RoboDK station: Example-03.d-Polishing Canadian Canoe - KUKA.rdk

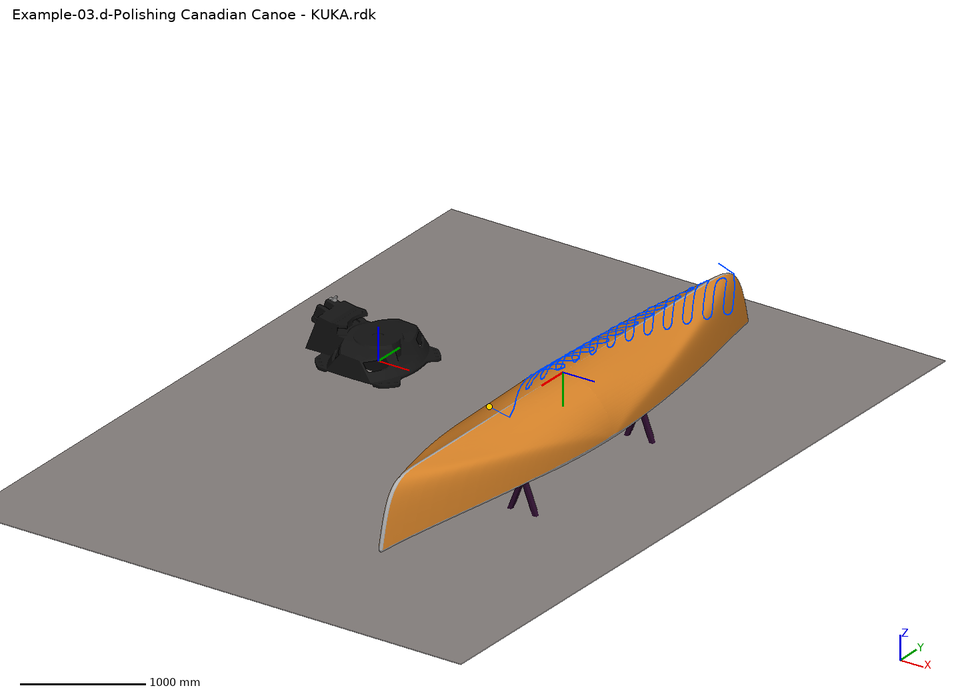
[picture v0: the station drawn from its stored meshes, robots at their saved joint values, targets as dots, program paths as lines]
Station Canoe Record Station final. Poses are relative to the parent item; angles as X-Y-Z fixed-axis rotations.
  - frame World at (0, 0, 0) mm
    - object Floor at (1290, -760, -10) mm, rotated rx 0 ry 0 rz 90 deg, size 6720 x 4800 x 9.6 mm, geometry from Floor.step
    - object Canoe Holder at (2372.71, -1561.9, -4.29) mm, rotated rx -180 ry 0 rz 0 deg, size 378 x 1657.8 x 756 mm, geometry from Canoe Holder.step
  - frame KUKA KR 100 R3500 press Base at (0, 0, 0) mm
    - robot KUKA KR 100 R3500 press: 6 axes, payload 100 kg, reach 3501 mm, repeatability 0.06 mm, weight 1240 kg
        joint limits [-185, -120, -120, -350, -122.5, -350] to [185, 70, 155, 350, 122.5, 350]; home [0, -90, 90, 0, 0, 0]; saved at [6.556, -77.694, 99.787, -0.648, 50.095, 7.142]
      - tool Sanding Tool, TCP at (0, 0, 140.65) mm, size 253.6 x 268.9 x 140.8 mm, geometry from Sanding Tool.step
  - frame Part at (2500, -1000, 1000) mm, rotated rx -90 ry 0 rz -90 deg
    - object Canadian Canoe at (0, 0, 0) mm, size 5096.7 x 583.7 x 963.7 mm, geometry from Canadian Canoe.step
    - object Polish Path 1 at (0, 0, 0) mm
  - machining project Polish Path 1 Settings: rotZ(0) | rotX(0)*rotY(0) | rotz(0) | ChangeTool(toolid) | onPathStart | PolishOn | onPoint | PolishOff | onFinish | SetRPM(%1) | SetTool(%1) | Extruder(%1) | default | default | OutOnMov(%1) | OutOffMov(%1) | onPathFinish | M_RunCode(%1)
  - program Polish (1259 instructions, listed below)
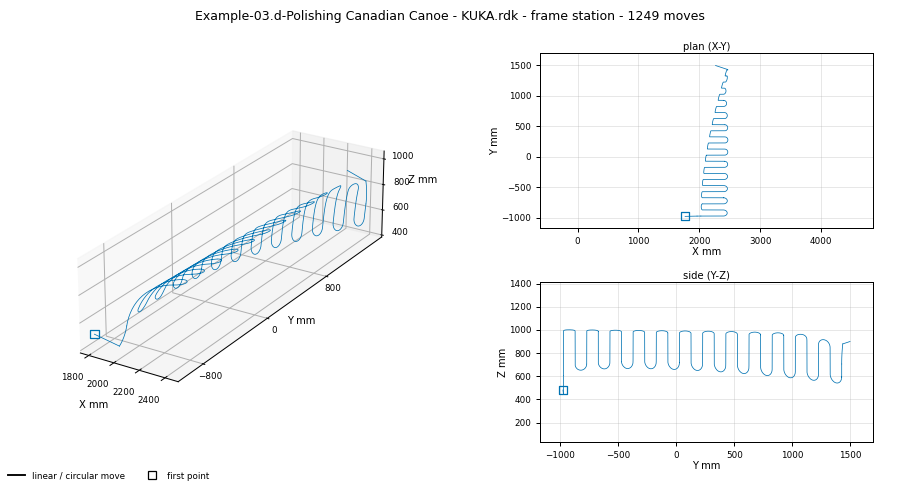
[picture p0: tool path of Example-03.d-Polishing Canadian Canoe - KUKA.rdk in frame station, 1249 of 1249 moves have a stored position in this frame; points joined in program order, loops and branches not executed]

--- program Polish (robot KUKA KR 100 R3500 press) ---
  Call ChangeTool(toolid)
  Smooth(1)
  Set Ref.: Part
  Set Tool: Sanding Tool
  Show Sanding Tool
  Set speed (200.0 mm/s)
  MoveJ 1 to (-21.87, 518.76, -734.4) mm, rotated rx 0 ry 10.84 rz 96.44 deg; joints [35.321, -70.266, 137.679, -138.31, 61.6, 158.371]
  MoveL 2 to (-21.87, 518.76, -734.4) mm, rotated rx 0 ry 10.84 rz 96.44 deg; joints [35.321, -70.266, 137.679, -138.31, 61.6, 158.371]
  Call PolishOn
  MoveL 3 to (-26.09, 556.13, -537.97) mm, rotated rx 0 ry 10.84 rz 96.44 deg; joints [31.728, -64.525, 130.322, -141.639, 59.446, 158.433]
  MoveC 4 to (-26.54, 477.64, -500.08) mm, rotated rx 0 ry 10.84 rz 96.44 deg; joints [31.115, -67.789, 128.968, -140.477, 55.681, 155.246] to (-26.66, 393.76, -476.39) mm, rotated rx 0 ry 10.84 rz 96.44 deg; joints [30.747, -71.291, 127.887, -138.729, 52.066, 151.749]
  MoveL 5 to (-26.66, 393.76, -476.39) mm, rotated rx 0 ry 10.84 rz 96.44 deg; joints [30.747, -71.291, 127.887, -138.729, 52.066, 151.749]
  MoveL 6 to (-26.66, 393.76, -476.39) mm, rotated rx 0 ry 10.84 rz 96.44 deg; joints [30.747, -71.291, 127.887, -138.729, 52.066, 151.749]
  Set speed (50.0 mm/s)
  MoveL 7 to (-26.66, 376.38, -472.76) mm, rotated rx 0 ry 12.85 rz 94.05 deg; joints [30.597, -72.582, 127.559, -137.347, 48.797, 152.34]
  MoveL 8 to (-26.66, 359.15, -468.51) mm, rotated rx 0 ry 14.9 rz 92.45 deg; joints [30.438, -73.793, 127.144, -135.658, 45.564, 151.886]
  MoveL 9 to (-26.66, 342.08, -463.65) mm, rotated rx 0 ry 16.96 rz 91.33 deg; joints [30.267, -74.917, 126.648, -133.634, 42.392, 150.663]
  MoveL 10 to (-26.66, 325.2, -458.16) mm, rotated rx 0 ry 19.04 rz 90.51 deg; joints [30.085, -75.951, 126.072, -131.226, 39.302, 148.785]
  MoveL 11 to (-26.66, 308.53, -452.07) mm, rotated rx 0 ry 21.12 rz 89.91 deg; joints [29.892, -76.889, 125.421, -128.37, 36.321, 146.284]
  MoveL 12 to (-26.66, 292.1, -445.38) mm, rotated rx 0 ry 23.2 rz 89.45 deg; joints [29.688, -77.729, 124.697, -124.985, 33.477, 143.138]
  MoveL 13 to (-26.66, 275.92, -438.09) mm, rotated rx 0 ry 25.28 rz 89.1 deg; joints [29.473, -78.472, 123.903, -120.973, 30.8, 139.286]
  MoveL 14 to (-26.66, 260.02, -430.23) mm, rotated rx 0 ry 27.37 rz 88.83 deg; joints [29.249, -79.115, 123.044, -116.23, 28.333, 134.648]
  MoveL 15 to (-26.66, 244.43, -421.8) mm, rotated rx 0 ry 29.45 rz 88.63 deg; joints [29.016, -79.659, 122.123, -110.659, 26.129, 129.146]
  MoveL 16 to (-26.66, 229.18, -412.82) mm, rotated rx 0 ry 31.53 rz 88.47 deg; joints [28.774, -80.105, 121.144, -104.187, 24.244, 122.718]
  MoveL 17 to (-26.66, 214.28, -403.3) mm, rotated rx 0 ry 33.61 rz 88.36 deg; joints [28.526, -80.455, 120.109, -96.804, 22.741, 115.363]
  MoveL 18 to (-26.66, 199.73, -393.26) mm, rotated rx 0 ry 35.69 rz 88.29 deg; joints [28.27, -80.711, 119.022, -88.615, 21.681, 107.193]
  MoveL 19 to (-26.66, 185.57, -382.7) mm, rotated rx 0 ry 37.76 rz 88.24 deg; joints [28.009, -80.875, 117.885, -79.876, 21.113, 98.467]
  MoveL 20 to (-26.66, 171.8, -371.63) mm, rotated rx 0 ry 39.84 rz 88.21 deg; joints [27.742, -80.951, 116.702, -70.965, 21.059, 89.568]
  MoveL 21 to (-26.66, 158.43, -360.06) mm, rotated rx 0 ry 41.92 rz 88.2 deg; joints [27.471, -80.94, 115.473, -62.307, 21.506, 80.922]
  MoveL 22 to (-26.66, 145.48, -348.01) mm, rotated rx 0 ry 44 rz 88.21 deg; joints [27.195, -80.847, 114.201, -54.254, 22.41, 72.884]
  MoveL 23 to (-26.66, 132.96, -335.48) mm, rotated rx 0 ry 46.08 rz 88.23 deg; joints [26.916, -80.673, 112.889, -47.021, 23.705, 65.671]
  MoveL 24 to (-26.66, 120.89, -322.49) mm, rotated rx 0 ry 48.17 rz 88.26 deg; joints [26.634, -80.422, 111.538, -40.68, 25.319, 59.356]
  MoveL 25 to (-26.66, 109.3, -309.06) mm, rotated rx 0 ry 50.26 rz 88.31 deg; joints [26.35, -80.098, 110.152, -35.208, 27.184, 53.915]
  MoveL 26 to (-26.66, 98.22, -295.23) mm, rotated rx 0 ry 52.34 rz 88.36 deg; joints [26.065, -79.703, 108.734, -30.523, 29.238, 49.268]
  MoveL 27 to (-26.66, 87.66, -281.03) mm, rotated rx 0 ry 54.43 rz 88.42 deg; joints [25.78, -79.242, 107.288, -26.513, 31.434, 45.305]
  MoveL 28 to (-26.66, 77.63, -266.46) mm, rotated rx 0 ry 56.51 rz 88.49 deg; joints [25.495, -78.717, 105.814, -23.071, 33.738, 41.916]
  MoveL 29 to (-26.66, 68.14, -251.54) mm, rotated rx 0 ry 58.59 rz 88.56 deg; joints [25.211, -78.131, 104.313, -20.1, 36.12, 39.008]
  MoveL 30 to (-26.66, 59.2, -236.29) mm, rotated rx 0 ry 60.67 rz 88.64 deg; joints [24.928, -77.488, 102.788, -17.519, 38.562, 36.499]
  MoveL 31 to (-26.66, 50.82, -220.71) mm, rotated rx 0 ry 62.76 rz 88.72 deg; joints [24.646, -76.789, 101.238, -15.262, 41.049, 34.323]
  MoveL 32 to (-26.66, 43.01, -204.84) mm, rotated rx 0 ry 64.84 rz 88.81 deg; joints [24.365, -76.038, 99.664, -13.273, 43.568, 32.426]
  MoveL 33 to (-26.66, 35.77, -188.67) mm, rotated rx 0 ry 66.93 rz 88.9 deg; joints [24.087, -75.236, 98.069, -11.508, 46.112, 30.763]
  MoveL 34 to (-26.66, 29.12, -172.23) mm, rotated rx 0 ry 69.03 rz 88.99 deg; joints [23.811, -74.386, 96.451, -9.931, 48.674, 29.299]
  MoveL 35 to (-26.66, 23.07, -155.55) mm, rotated rx 0 ry 71.12 rz 89.09 deg; joints [23.539, -73.49, 94.814, -8.515, 51.247, 28.008]
  MoveL 36 to (-26.66, 17.65, -138.69) mm, rotated rx 0 ry 73.21 rz 89.19 deg; joints [23.27, -72.554, 93.162, -7.236, 53.821, 26.866]
  MoveL 37 to (-26.66, 12.84, -121.65) mm, rotated rx 0 ry 75.3 rz 89.29 deg; joints [23.005, -71.578, 91.496, -6.073, 56.395, 25.853]
  MoveL 38 to (-26.66, 8.67, -104.47) mm, rotated rx 0 ry 77.39 rz 89.39 deg; joints [22.744, -70.564, 89.814, -5.01, 58.966, 24.952]
  MoveL 39 to (-26.66, 8.67, -104.47) mm, rotated rx 0 ry 77.39 rz 89.39 deg; joints [22.744, -70.564, 89.814, -5.01, 58.966, 24.952]
  MoveL 40 to (-27.51, 6.41, -93.75) mm, rotated rx 0 ry 78.68 rz 89.45 deg; joints [22.566, -69.932, 88.785, -4.39, 60.546, 24.425]
  MoveL 41 to (-30.02, 4.45, -83.22) mm, rotated rx 0 ry 79.94 rz 89.51 deg; joints [22.359, -69.329, 87.813, -3.806, 62.065, 23.908]
  MoveL 42 to (-34.12, 2.8, -73.18) mm, rotated rx 0 ry 81.12 rz 89.56 deg; joints [22.129, -68.772, 86.925, -3.274, 63.484, 23.411]
  MoveL 43 to (-39.8, 1.48, -63.88) mm, rotated rx 0 ry 82.19 rz 89.6 deg; joints [21.88, -68.28, 86.145, -2.802, 64.765, 22.939]
  MoveL 44 to (-43.22, 0.94, -59.64) mm, rotated rx 0 ry 82.68 rz 89.62 deg; joints [21.751, -68.066, 85.808, -2.593, 65.337, 22.715]
  MoveL 45 to (-47.01, 0.48, -55.73) mm, rotated rx 0 ry 83.12 rz 89.64 deg; joints [21.618, -67.878, 85.512, -2.405, 65.854, 22.499]
  MoveL 46 to (-51.17, 0.09, -52.22) mm, rotated rx 0 ry 83.51 rz 89.65 deg; joints [21.485, -67.72, 85.263, -2.24, 66.307, 22.295]
  MoveL 47 to (-55.67, -0.22, -49.18) mm, rotated rx 0 ry 83.85 rz 89.67 deg; joints [21.351, -67.597, 85.069, -2.099, 66.686, 22.102]
  MoveL 48 to (-60.51, -0.46, -46.68) mm, rotated rx 0 ry 84.11 rz 89.67 deg; joints [21.219, -67.513, 84.934, -1.984, 66.981, 21.922]
  MoveL 49 to (-65.61, -0.62, -44.79) mm, rotated rx 0 ry 84.3 rz 89.68 deg; joints [21.089, -67.474, 84.867, -1.899, 67.181, 21.759]
  MoveL 50 to (-70.92, -0.71, -43.6) mm, rotated rx 0 ry 84.4 rz 89.68 deg; joints [20.965, -67.482, 84.872, -1.845, 67.278, 21.614]
  MoveL 51 to (-76.36, -0.72, -43.15) mm, rotated rx 0 ry 84.42 rz 89.67 deg; joints [20.847, -67.54, 84.952, -1.823, 67.264, 21.49]
  MoveL 52 to (-81.8, -0.66, -43.46) mm, rotated rx 0 ry 84.34 rz 89.66 deg; joints [20.74, -67.648, 85.106, -1.833, 67.137, 21.389]
  MoveL 53 to (-87.14, -0.52, -44.52) mm, rotated rx 0 ry 84.17 rz 89.65 deg; joints [20.643, -67.803, 85.332, -1.873, 66.903, 21.312]
  MoveL 54 to (-92.3, -0.3, -46.28) mm, rotated rx 0 ry 83.92 rz 89.62 deg; joints [20.56, -68, 85.622, -1.941, 66.568, 21.261]
  MoveL 55 to (-97.19, -0.01, -48.67) mm, rotated rx 0 ry 83.6 rz 89.6 deg; joints [20.49, -68.234, 85.967, -2.035, 66.143, 21.236]
  MoveL 56 to (-101.76, 0.37, -51.62) mm, rotated rx 0 ry 83.21 rz 89.57 deg; joints [20.432, -68.498, 86.359, -2.151, 65.641, 21.234]
  MoveL 57 to (-105.99, 0.82, -55.04) mm, rotated rx 0 ry 82.77 rz 89.53 deg; joints [20.388, -68.786, 86.79, -2.287, 65.073, 21.257]
  MoveL 58 to (-109.84, 1.36, -58.88) mm, rotated rx 0 ry 82.29 rz 89.49 deg; joints [20.357, -69.093, 87.252, -2.441, 64.45, 21.302]
  MoveL 59 to (-113.32, 1.98, -63.07) mm, rotated rx 0 ry 81.76 rz 89.45 deg; joints [20.338, -69.415, 87.739, -2.611, 63.78, 21.37]
  MoveL 60 to (-119.09, 3.46, -72.25) mm, rotated rx 0 ry 80.62 rz 89.36 deg; joints [20.334, -70.086, 88.764, -2.994, 62.336, 21.568]
  MoveL 61 to (-123.26, 5.27, -82.23) mm, rotated rx 0 ry 79.41 rz 89.27 deg; joints [20.374, -70.773, 89.829, -3.428, 60.794, 21.85]
  MoveL 62 to (-125.8, 7.38, -92.7) mm, rotated rx 0 ry 78.14 rz 89.17 deg; joints [20.457, -71.455, 90.903, -3.911, 59.199, 22.212]
  MoveL 63 to (-126.66, 9.76, -103.38) mm, rotated rx 0 ry 76.86 rz 89.08 deg; joints [20.58, -72.113, 91.96, -4.437, 57.594, 22.653]
  MoveL 64 to (-126.66, 9.76, -103.38) mm, rotated rx 0 ry 76.86 rz 89.08 deg; joints [20.58, -72.113, 91.96, -4.437, 57.594, 22.653]
  MoveL 65 to (-126.66, 17.22, -131.53) mm, rotated rx 0 ry 73.48 rz 88.86 deg; joints [20.967, -73.761, 94.694, -6.011, 53.356, 24.056]
  MoveL 66 to (-126.66, 26.34, -159.24) mm, rotated rx 0 ry 70.1 rz 88.67 deg; joints [21.365, -75.303, 97.386, -7.878, 49.121, 25.774]
  MoveL 67 to (-126.66, 37.07, -186.38) mm, rotated rx 0 ry 66.74 rz 88.5 deg; joints [21.775, -76.728, 100.027, -10.127, 44.908, 27.89]
  MoveL 68 to (-126.66, 49.36, -212.8) mm, rotated rx 0 ry 63.4 rz 88.36 deg; joints [22.195, -78.024, 102.61, -12.882, 40.74, 30.524]
  MoveL 69 to (-126.66, 63.15, -238.44) mm, rotated rx 0 ry 60.06 rz 88.26 deg; joints [22.623, -79.183, 105.132, -16.314, 36.644, 33.846]
  MoveL 70 to (-126.66, 78.41, -263.23) mm, rotated rx 0 ry 56.73 rz 88.19 deg; joints [23.059, -80.193, 107.588, -20.673, 32.668, 38.1]
  MoveL 71 to (-126.66, 95.1, -287.12) mm, rotated rx 0 ry 53.42 rz 88.17 deg; joints [23.501, -81.043, 109.974, -26.314, 28.89, 43.635]
  MoveL 72 to (-126.66, 113.18, -310.05) mm, rotated rx 0 ry 50.1 rz 88.21 deg; joints [23.948, -81.719, 112.284, -33.726, 25.435, 50.931]
  MoveL 73 to (-126.66, 132.55, -331.89) mm, rotated rx 0 ry 46.8 rz 88.32 deg; joints [24.398, -82.205, 114.505, -43.444, 22.513, 60.518]
  MoveL 74 to (-126.66, 153.11, -352.55) mm, rotated rx 0 ry 43.5 rz 88.51 deg; joints [24.847, -82.489, 116.626, -55.814, 20.415, 72.728]
  MoveL 75 to (-126.66, 174.81, -371.99) mm, rotated rx 0 ry 40.22 rz 88.81 deg; joints [25.293, -82.556, 118.64, -70.412, 19.477, 87.12]
  MoveL 76 to (-126.66, 197.6, -390.16) mm, rotated rx 0 ry 36.95 rz 89.25 deg; joints [25.735, -82.393, 120.536, -85.632, 19.933, 102.065]
  MoveL 77 to (-126.66, 221.41, -407.03) mm, rotated rx 0 ry 33.68 rz 89.87 deg; joints [26.17, -81.987, 122.306, -99.424, 21.768, 115.479]
  MoveL 78 to (-126.66, 246.16, -422.53) mm, rotated rx 0 ry 30.43 rz 90.72 deg; joints [26.595, -81.327, 123.935, -110.611, 24.74, 126.138]
  MoveL 79 to (-126.66, 271.73, -436.59) mm, rotated rx 0 ry 27.19 rz 91.88 deg; joints [27.005, -80.405, 125.409, -119.146, 28.539, 133.925]
  MoveL 80 to (-126.66, 298.05, -449.17) mm, rotated rx 0 ry 23.97 rz 93.45 deg; joints [27.397, -79.22, 126.718, -125.536, 32.912, 139.252]
  MoveL 81 to (-126.66, 298.05, -449.17) mm, rotated rx 0 ry 23.97 rz 93.45 deg; joints [27.397, -79.22, 126.718, -125.536, 32.912, 139.252]
  MoveL 82 to (-127.57, 307.4, -453.24) mm, rotated rx 0 ry 22.87 rz 94.13 deg; joints [27.505, -78.761, 127.15, -127.373, 34.523, 140.591]
  MoveL 83 to (-130.27, 316.51, -457.06) mm, rotated rx 0 ry 21.82 rz 94.91 deg; joints [27.562, -78.32, 127.583, -129.005, 36.088, 141.626]
  MoveL 84 to (-134.68, 325.06, -460.55) mm, rotated rx 0 ry 20.87 rz 95.71 deg; joints [27.561, -77.916, 128.01, -130.458, 37.553, 142.427]
  MoveL 85 to (-140.71, 332.73, -463.63) mm, rotated rx 0 ry 19.99 rz 96.43 deg; joints [27.5, -77.568, 128.431, -131.809, 38.881, 143.152]
  MoveL 86 to (-144.29, 336.12, -464.99) mm, rotated rx 0 ry 19.57 rz 96.71 deg; joints [27.445, -77.419, 128.64, -132.482, 39.488, 143.56]
  MoveL 87 to (-148.2, 339.15, -466.21) mm, rotated rx 0 ry 19.15 rz 96.9 deg; joints [27.372, -77.288, 128.85, -133.177, 40.06, 144.046]
  MoveL 88 to (-152.44, 341.79, -467.28) mm, rotated rx 0 ry 18.73 rz 96.99 deg; joints [27.282, -77.177, 129.06, -133.911, 40.6, 144.643]
  MoveL 89 to (-156.95, 344, -468.2) mm, rotated rx 0 ry 18.31 rz 96.96 deg; joints [27.174, -77.084, 129.272, -134.688, 41.108, 145.369]
  MoveL 90 to (-161.69, 345.73, -468.95) mm, rotated rx 0 ry 17.88 rz 96.8 deg; joints [27.051, -77.014, 129.481, -135.496, 41.579, 146.218]
  MoveL 91 to (-166.61, 346.96, -469.52) mm, rotated rx 0 ry 17.46 rz 96.53 deg; joints [26.913, -76.969, 129.683, -136.309, 42, 147.154]
  MoveL 92 to (-171.65, 347.66, -469.91) mm, rotated rx 0 ry 17.09 rz 96.18 deg; joints [26.765, -76.954, 129.872, -137.083, 42.346, 148.113]
  MoveL 93 to (-176.74, 347.81, -470.12) mm, rotated rx 0 ry 16.8 rz 95.79 deg; joints [26.61, -76.976, 130.039, -137.76, 42.582, 149.006]
  MoveL 94 to (-181.84, 347.4, -470.15) mm, rotated rx 0 ry 16.61 rz 95.41 deg; joints [26.452, -77.042, 130.179, -138.295, 42.677, 149.752]
  MoveL 95 to (-186.86, 346.44, -470) mm, rotated rx 0 ry 16.56 rz 95.08 deg; joints [26.294, -77.157, 130.285, -138.647, 42.603, 150.279]
  MoveL 96 to (-191.75, 344.95, -469.68) mm, rotated rx 0 ry 16.67 rz 94.83 deg; joints [26.14, -77.321, 130.355, -138.794, 42.346, 150.54]
  MoveL 97 to (-196.44, 342.96, -469.2) mm, rotated rx 0 ry 16.92 rz 94.67 deg; joints [25.992, -77.532, 130.385, -138.725, 41.904, 150.518]
  MoveL 98 to (-200.89, 340.51, -468.56) mm, rotated rx 0 ry 17.33 rz 94.6 deg; joints [25.851, -77.786, 130.377, -138.441, 41.29, 150.216]
  MoveL 99 to (-205.06, 337.66, -467.76) mm, rotated rx 0 ry 17.86 rz 94.6 deg; joints [25.717, -78.075, 130.33, -137.951, 40.524, 149.658]
  MoveL 100 to (-212.46, 330.89, -465.7) mm, rotated rx 0 ry 19.23 rz 94.73 deg; joints [25.472, -78.721, 130.131, -136.411, 38.646, 147.908]
  MoveL 101 to (-218.45, 323.03, -463.03) mm, rotated rx 0 ry 20.86 rz 94.87 deg; joints [25.253, -79.402, 129.811, -134.269, 36.508, 145.573]
  MoveL 102 to (-222.9, 314.4, -459.75) mm, rotated rx 0 ry 22.54 rz 94.9 deg; joints [25.059, -80.059, 129.399, -131.722, 34.323, 142.947]
  MoveL 103 to (-225.67, 305.32, -455.94) mm, rotated rx 0 ry 24.16 rz 94.76 deg; joints [24.891, -80.653, 128.925, -128.966, 32.247, 140.254]
  MoveL 104 to (-226.66, 296.05, -451.69) mm, rotated rx 0 ry 25.64 rz 94.48 deg; joints [24.753, -81.164, 128.41, -126.131, 30.355, 137.613]
  MoveL 105 to (-226.66, 296.05, -451.69) mm, rotated rx 0 ry 25.64 rz 94.48 deg; joints [24.753, -81.164, 128.41, -126.131, 30.355, 137.613]
  MoveL 106 to (-226.66, 270.18, -438.28) mm, rotated rx 0 ry 29.16 rz 93.21 deg; joints [24.38, -82.288, 126.92, -117.969, 25.867, 130.316]
  MoveL 107 to (-226.66, 245.16, -423.4) mm, rotated rx 0 ry 32.32 rz 91.9 deg; joints [23.966, -83.105, 125.374, -108.343, 22.255, 121.554]
  MoveL 108 to (-226.66, 221.07, -407.26) mm, rotated rx 0 ry 35.36 rz 90.79 deg; joints [23.538, -83.661, 123.728, -96.225, 19.574, 110.144]
  MoveL 109 to (-226.66, 197.82, -389.81) mm, rotated rx 0 ry 38.4 rz 89.91 deg; joints [23.104, -83.977, 121.962, -81.528, 18.063, 96]
  MoveL 110 to (-226.66, 175.5, -371.14) mm, rotated rx 0 ry 41.45 rz 89.24 deg; joints [22.669, -84.067, 120.08, -65.719, 17.94, 80.615]
  MoveL 111 to (-226.66, 154.2, -351.29) mm, rotated rx 0 ry 44.51 rz 88.74 deg; joints [22.236, -83.94, 118.092, -51.11, 19.167, 66.33]
  MoveL 112 to (-226.66, 134.01, -330.36) mm, rotated rx 0 ry 47.59 rz 88.38 deg; joints [21.807, -83.612, 116.007, -39.179, 21.459, 54.645]
  MoveL 113 to (-226.66, 114.99, -308.38) mm, rotated rx 0 ry 50.69 rz 88.14 deg; joints [21.385, -83.094, 113.834, -30.079, 24.47, 45.735]
  MoveL 114 to (-226.66, 97.2, -285.42) mm, rotated rx 0 ry 53.8 rz 88 deg; joints [20.97, -82.4, 111.579, -23.269, 27.933, 39.072]
  MoveL 115 to (-226.66, 80.67, -261.51) mm, rotated rx 0 ry 56.93 rz 87.94 deg; joints [20.565, -81.541, 109.247, -18.143, 31.677, 34.061]
  MoveL 116 to (-226.66, 65.47, -236.71) mm, rotated rx 0 ry 60.09 rz 87.96 deg; joints [20.168, -80.528, 106.841, -14.214, 35.601, 30.228]
  MoveL 117 to (-226.66, 51.64, -211.07) mm, rotated rx 0 ry 63.27 rz 88.03 deg; joints [19.782, -79.372, 104.366, -11.151, 39.636, 27.249]
  MoveL 118 to (-226.66, 39.23, -184.63) mm, rotated rx 0 ry 66.48 rz 88.16 deg; joints [19.406, -78.081, 101.827, -8.724, 43.736, 24.898]
  MoveL 119 to (-226.66, 28.33, -157.54) mm, rotated rx 0 ry 69.69 rz 88.34 deg; joints [19.044, -76.67, 99.236, -6.78, 47.865, 23.026]
  MoveL 120 to (-226.66, 18.99, -129.94) mm, rotated rx 0 ry 72.93 rz 88.56 deg; joints [18.696, -75.147, 96.597, -5.195, 52.015, 21.515]
  MoveL 121 to (-226.66, 11.24, -101.9) mm, rotated rx 0 ry 76.19 rz 88.82 deg; joints [18.36, -73.52, 93.91, -3.883, 56.181, 20.285]
  MoveL 122 to (-226.66, 11.24, -101.9) mm, rotated rx 0 ry 76.19 rz 88.82 deg; joints [18.36, -73.52, 93.91, -3.883, 56.181, 20.285]
  MoveL 123 to (-227.52, 8.78, -91.34) mm, rotated rx 0 ry 77.4 rz 88.93 deg; joints [18.22, -72.9, 92.915, -3.447, 57.721, 19.867]
  MoveL 124 to (-230.03, 6.62, -80.99) mm, rotated rx 0 ry 78.57 rz 89.03 deg; joints [18.048, -72.307, 91.971, -3.043, 59.197, 19.449]
  MoveL 125 to (-234.15, 4.79, -71.12) mm, rotated rx 0 ry 79.66 rz 89.13 deg; joints [17.849, -71.758, 91.106, -2.682, 60.569, 19.04]
  MoveL 126 to (-239.84, 3.29, -62.01) mm, rotated rx 0 ry 80.65 rz 89.22 deg; joints [17.628, -71.271, 90.345, -2.369, 61.796, 18.645]
  MoveL 127 to (-243.26, 2.67, -57.85) mm, rotated rx 0 ry 81.09 rz 89.26 deg; joints [17.511, -71.059, 90.014, -2.234, 62.338, 18.455]
  MoveL 128 to (-247.05, 2.13, -54.03) mm, rotated rx 0 ry 81.48 rz 89.3 deg; joints [17.39, -70.872, 89.724, -2.113, 62.823, 18.27]
  MoveL 129 to (-251.2, 1.68, -50.61) mm, rotated rx 0 ry 81.82 rz 89.34 deg; joints [17.266, -70.715, 89.479, -2.009, 63.243, 18.092]
  MoveL 130 to (-255.68, 1.31, -47.64) mm, rotated rx 0 ry 82.11 rz 89.37 deg; joints [17.139, -70.591, 89.285, -1.923, 63.589, 17.922]
  MoveL 131 to (-260.49, 1.03, -45.2) mm, rotated rx 0 ry 82.33 rz 89.39 deg; joints [17.012, -70.504, 89.148, -1.854, 63.852, 17.761]
  MoveL 132 to (-265.54, 0.83, -43.36) mm, rotated rx 0 ry 82.47 rz 89.41 deg; joints [16.886, -70.46, 89.074, -1.804, 64.022, 17.61]
  MoveL 133 to (-270.8, 0.73, -42.18) mm, rotated rx 0 ry 82.54 rz 89.42 deg; joints [16.762, -70.46, 89.067, -1.773, 64.092, 17.472]
  MoveL 134 to (-276.18, 0.72, -41.71) mm, rotated rx 0 ry 82.53 rz 89.42 deg; joints [16.642, -70.507, 89.131, -1.761, 64.058, 17.349]
  MoveL 135 to (-281.57, 0.81, -41.96) mm, rotated rx 0 ry 82.43 rz 89.41 deg; joints [16.528, -70.601, 89.264, -1.768, 63.918, 17.242]
  MoveL 136 to (-286.88, 1, -42.92) mm, rotated rx 0 ry 82.25 rz 89.39 deg; joints [16.423, -70.739, 89.464, -1.792, 63.677, 17.153]
  MoveL 137 to (-291.99, 1.28, -44.55) mm, rotated rx 0 ry 82 rz 89.36 deg; joints [16.328, -70.916, 89.724, -1.833, 63.343, 17.083]
  MoveL 138 to (-296.87, 1.66, -46.8) mm, rotated rx 0 ry 81.68 rz 89.33 deg; joints [16.244, -71.128, 90.036, -1.887, 62.927, 17.032]
  MoveL 139 to (-301.46, 2.13, -49.6) mm, rotated rx 0 ry 81.31 rz 89.28 deg; joints [16.17, -71.37, 90.396, -1.954, 62.436, 17]
  MoveL 140 to (-305.71, 2.7, -52.88) mm, rotated rx 0 ry 80.88 rz 89.23 deg; joints [16.108, -71.637, 90.794, -2.033, 61.884, 16.986]
  MoveL 141 to (-309.61, 3.36, -56.58) mm, rotated rx 0 ry 80.42 rz 89.18 deg; joints [16.057, -71.922, 91.223, -2.122, 61.28, 16.992]
  MoveL 142 to (-313.12, 4.12, -60.63) mm, rotated rx 0 ry 79.92 rz 89.12 deg; joints [16.017, -72.223, 91.677, -2.22, 60.634, 17.015]
  MoveL 143 to (-318.97, 5.89, -69.57) mm, rotated rx 0 ry 78.86 rz 89 deg; joints [15.97, -72.854, 92.64, -2.443, 59.244, 17.116]
  MoveL 144 to (-323.21, 7.99, -79.34) mm, rotated rx 0 ry 77.72 rz 88.86 deg; joints [15.966, -73.504, 93.645, -2.702, 57.769, 17.287]
  MoveL 145 to (-325.79, 10.39, -89.6) mm, rotated rx 0 ry 76.56 rz 88.73 deg; joints [16.005, -74.152, 94.663, -2.995, 56.253, 17.529]
  MoveL 146 to (-326.66, 13.03, -100.1) mm, rotated rx 0 ry 75.39 rz 88.61 deg; joints [16.087, -74.781, 95.668, -3.324, 54.732, 17.842]
  MoveL 147 to (-326.66, 13.03, -100.1) mm, rotated rx 0 ry 75.39 rz 88.61 deg; joints [16.087, -74.781, 95.668, -3.324, 54.732, 17.842]
  MoveL 148 to (-326.66, 21.62, -129.56) mm, rotated rx 0 ry 72.14 rz 88.3 deg; joints [16.384, -76.457, 98.434, -4.419, 50.483, 18.938]
  MoveL 149 to (-326.66, 31.86, -158.52) mm, rotated rx 0 ry 68.93 rz 88.05 deg; joints [16.696, -78.02, 101.142, -5.79, 46.265, 20.303]
  MoveL 150 to (-326.66, 43.68, -186.84) mm, rotated rx 0 ry 65.77 rz 87.87 deg; joints [17.024, -79.46, 103.785, -7.521, 42.095, 22.014]
  MoveL 151 to (-326.66, 57.07, -214.48) mm, rotated rx 0 ry 62.61 rz 87.76 deg; joints [17.37, -80.777, 106.377, -9.76, 37.937, 24.211]
  MoveL 152 to (-326.66, 71.99, -241.41) mm, rotated rx 0 ry 59.46 rz 87.73 deg; joints [17.731, -81.959, 108.912, -12.681, 33.824, 27.066]
  MoveL 153 to (-326.66, 88.43, -267.6) mm, rotated rx 0 ry 56.34 rz 87.78 deg; joints [18.11, -82.994, 111.386, -16.559, 29.804, 30.844]
  MoveL 154 to (-326.66, 106.3, -292.91) mm, rotated rx 0 ry 53.25 rz 87.94 deg; joints [18.503, -83.867, 113.783, -21.795, 25.967, 35.936]
  MoveL 155 to (-326.66, 125.5, -317.22) mm, rotated rx 0 ry 50.19 rz 88.22 deg; joints [18.91, -84.564, 116.098, -28.995, 22.426, 42.935]
  MoveL 156 to (-326.66, 145.96, -340.48) mm, rotated rx 0 ry 47.16 rz 88.64 deg; joints [19.33, -85.073, 118.326, -38.968, 19.38, 52.635]
  MoveL 157 to (-326.66, 167.61, -362.62) mm, rotated rx 0 ry 44.14 rz 89.22 deg; joints [19.761, -85.38, 120.461, -52.426, 17.151, 65.732]
  MoveL 158 to (-326.66, 190.17, -383.4) mm, rotated rx 0 ry 41.15 rz 89.97 deg; joints [20.197, -85.471, 122.48, -68.918, 16.152, 81.766]
  MoveL 159 to (-326.66, 201.28, -392.87) mm, rotated rx 0 ry 39.72 rz 90.38 deg; joints [20.406, -85.435, 123.41, -77.359, 16.195, 89.951]
  MoveL 160 to (-326.66, 212.12, -401.66) mm, rotated rx 0 ry 38.32 rz 90.81 deg; joints [20.605, -85.35, 124.282, -85.411, 16.568, 97.738]
  MoveL 161 to (-326.66, 222.63, -409.76) mm, rotated rx 0 ry 36.96 rz 91.23 deg; joints [20.794, -85.221, 125.101, -92.845, 17.223, 104.906]
  MoveL 162 to (-326.66, 232.74, -417.18) mm, rotated rx 0 ry 35.62 rz 91.63 deg; joints [20.97, -85.053, 125.869, -99.575, 18.105, 111.38]
  MoveL 163 to (-326.66, 242.39, -423.92) mm, rotated rx 0 ry 34.28 rz 91.99 deg; joints [21.131, -84.849, 126.591, -105.63, 19.166, 117.202]
  MoveL 164 to (-326.66, 251.51, -429.98) mm, rotated rx 0 ry 32.92 rz 92.29 deg; joints [21.274, -84.614, 127.272, -111.099, 20.372, 122.48]
  MoveL 165 to (-326.66, 260.05, -435.37) mm, rotated rx 0 ry 31.53 rz 92.48 deg; joints [21.4, -84.35, 127.917, -116.095, 21.703, 127.341]
  MoveL 166 to (-326.66, 268.03, -440.12) mm, rotated rx 0 ry 30.09 rz 92.56 deg; joints [21.506, -84.056, 128.534, -120.728, 23.159, 131.917]
  MoveL 167 to (-326.66, 275.46, -444.29) mm, rotated rx 0 ry 28.57 rz 92.5 deg; joints [21.592, -83.733, 129.125, -125.047, 24.738, 136.271]
  MoveL 168 to (-326.66, 282.36, -447.93) mm, rotated rx 0 ry 26.99 rz 92.29 deg; joints [21.66, -83.377, 129.693, -129.092, 26.453, 140.459]
  MoveL 169 to (-326.66, 282.36, -447.93) mm, rotated rx 0 ry 26.99 rz 92.29 deg; joints [21.66, -83.377, 129.693, -129.092, 26.453, 140.459]
  MoveL 170 to (-326.94, 287.31, -450.39) mm, rotated rx 0 ry 25.72 rz 92 deg; joints [21.69, -83.085, 130.119, -132.038, 27.859, 143.599]
  MoveL 171 to (-327.75, 292.26, -452.71) mm, rotated rx 0 ry 24.31 rz 91.56 deg; joints [21.696, -82.758, 130.567, -135.044, 29.444, 146.906]
  MoveL 172 to (-329.09, 297.17, -454.86) mm, rotated rx 0 ry 22.79 rz 90.94 deg; joints [21.675, -82.391, 131.03, -138.048, 31.215, 150.347]
  MoveL 173 to (-330.91, 301.99, -456.81) mm, rotated rx 0 ry 21.17 rz 90.13 deg; joints [21.629, -81.985, 131.495, -140.95, 33.145, 153.847]
  MoveL 174 to (-333.19, 306.67, -458.54) mm, rotated rx 0 ry 19.51 rz 89.1 deg; joints [21.559, -81.545, 131.948, -143.66, 35.189, 157.333]
  MoveL 175 to (-335.89, 311.18, -460.04) mm, rotated rx 0 ry 17.87 rz 87.87 deg; joints [21.468, -81.081, 132.376, -146.107, 37.277, 160.742]
  MoveL 176 to (-339.01, 315.49, -461.32) mm, rotated rx 0 ry 16.31 rz 86.47 deg; joints [21.36, -80.611, 132.768, -148.25, 39.327, 164.022]
  MoveL 177 to (-342.49, 319.53, -462.37) mm, rotated rx 0 ry 14.88 rz 84.94 deg; joints [21.237, -80.153, 133.117, -150.077, 41.257, 167.129]
  MoveL 178 to (-346.31, 323.27, -463.21) mm, rotated rx 0 ry 13.41 rz 82.89 deg; joints [21.091, -79.668, 133.453, -151.867, 43.277, 170.673]
  MoveL 179 to (-350.44, 326.66, -463.83) mm, rotated rx 0 ry 12.04 rz 80.41 deg; joints [20.928, -79.194, 133.758, -153.486, 45.22, 174.47]
  MoveL 180 to (-354.87, 329.66, -464.26) mm, rotated rx 0 ry 10.88 rz 77.74 deg; joints [20.757, -78.771, 134.016, -154.834, 46.912, 178.199]
  MoveL 181 to (-359.55, 332.21, -464.52) mm, rotated rx 0 ry 9.96 rz 75.08 deg; joints [20.58, -78.419, 134.232, -155.932, 48.306, 181.702]
  MoveL 182 to (-364.46, 334.24, -464.62) mm, rotated rx 0 ry 9.26 rz 72.59 deg; joints [20.399, -78.147, 134.409, -156.818, 49.395, 184.844]
  MoveL 183 to (-369.53, 335.7, -464.58) mm, rotated rx 0 ry 8.77 rz 70.44 deg; joints [20.217, -77.959, 134.555, -157.528, 50.19, 187.5]
  MoveL 184 to (-374.71, 336.52, -464.42) mm, rotated rx 0 ry 8.45 rz 68.72 deg; joints [20.035, -77.853, 134.673, -158.093, 50.717, 189.594]
  MoveL 185 to (-379.92, 336.69, -464.16) mm, rotated rx 0 ry 8.28 rz 67.52 deg; joints [19.855, -77.827, 134.768, -158.535, 50.994, 191.069]
  MoveL 186 to (-385.04, 336.19, -463.81) mm, rotated rx 0 ry 8.23 rz 66.87 deg; joints [19.681, -77.878, 134.839, -158.866, 51.039, 191.904]
  MoveL 187 to (-389.95, 335.08, -463.38) mm, rotated rx 0 ry 8.3 rz 66.76 deg; joints [19.516, -77.998, 134.887, -159.091, 50.874, 192.117]
  MoveL 188 to (-394.58, 333.42, -462.88) mm, rotated rx 0 ry 8.48 rz 67.13 deg; joints [19.364, -78.18, 134.914, -159.216, 50.515, 191.764]
  MoveL 189 to (-398.93, 331.27, -462.33) mm, rotated rx 0 ry 8.76 rz 67.94 deg; joints [19.222, -78.419, 134.918, -159.242, 49.972, 190.901]
  MoveL 190 to (-406.78, 325.7, -461.04) mm, rotated rx 0 ry 9.65 rz 70.64 deg; joints [18.976, -79.057, 134.856, -158.971, 48.317, 187.834]
  MoveL 191 to (-413.38, 318.81, -459.48) mm, rotated rx 0 ry 11.07 rz 74.34 deg; joints [18.782, -79.891, 134.678, -158.164, 45.857, 183.333]
  MoveL 192 to (-418.72, 310.96, -457.58) mm, rotated rx 0 ry 13.15 rz 78.48 deg; joints [18.642, -80.899, 134.349, -156.611, 42.506, 177.789]
  MoveL 193 to (-422.83, 302.26, -455.17) mm, rotated rx 0 ry 16 rz 82.45 deg; joints [18.55, -82.04, 133.819, -153.972, 38.224, 171.452]
  MoveL 194 to (-425.56, 292.93, -452.13) mm, rotated rx 0 ry 19.24 rz 85.44 deg; joints [18.485, -83.146, 133.108, -150.269, 33.608, 165.089]
  MoveL 195 to (-426.36, 287.77, -450.23) mm, rotated rx 0 ry 20.9 rz 86.51 deg; joints [18.455, -83.66, 132.692, -148.031, 31.313, 161.924]
  MoveL 196 to (-426.66, 282.26, -448.03) mm, rotated rx 0 ry 22.74 rz 87.55 deg; joints [18.437, -84.169, 132.197, -145.135, 28.867, 158.176]
  MoveL 197 to (-426.66, 282.26, -448.03) mm, rotated rx 0 ry 22.74 rz 87.55 deg; joints [18.437, -84.169, 132.197, -145.135, 28.867, 158.176]
  MoveL 198 to (-426.66, 270.66, -442.69) mm, rotated rx 0 ry 26.62 rz 89.24 deg; joints [18.397, -85.071, 131.045, -137.33, 24.077, 149.056]
  MoveL 199 to (-426.66, 267.36, -441) mm, rotated rx 0 ry 27.67 rz 89.6 deg; joints [18.379, -85.282, 130.705, -134.713, 22.867, 146.175]
  MoveL 200 to (-426.66, 263.49, -438.92) mm, rotated rx 0 ry 28.88 rz 89.96 deg; joints [18.354, -85.506, 130.302, -131.423, 21.548, 142.627]
  MoveL 201 to (-426.66, 259.04, -436.39) mm, rotated rx 0 ry 30.19 rz 90.29 deg; joints [18.32, -85.73, 129.84, -127.389, 20.184, 138.36]
  MoveL 202 to (-426.66, 254.01, -433.38) mm, rotated rx 0 ry 31.58 rz 90.58 deg; joints [18.274, -85.946, 129.323, -122.561, 18.841, 133.338]
  MoveL 203 to (-426.66, 248.41, -429.84) mm, rotated rx 0 ry 33.01 rz 90.8 deg; joints [18.216, -86.146, 128.757, -116.923, 17.586, 127.558]
  MoveL 204 to (-426.66, 242.23, -425.71) mm, rotated rx 0 ry 34.44 rz 90.94 deg; joints [18.144, -86.322, 128.15, -110.508, 16.476, 121.059]
  MoveL 205 to (-426.66, 235.47, -420.96) mm, rotated rx 0 ry 35.85 rz 90.99 deg; joints [18.056, -86.473, 127.505, -103.397, 15.554, 113.922]
  MoveL 206 to (-426.66, 228.14, -415.53) mm, rotated rx 0 ry 37.23 rz 90.95 deg; joints [17.952, -86.595, 126.825, -95.701, 14.846, 106.257]
  MoveL 207 to (-426.66, 220.24, -409.38) mm, rotated rx 0 ry 38.57 rz 90.83 deg; joints [17.832, -86.687, 126.109, -87.551, 14.372, 98.19]
  MoveL 208 to (-426.66, 211.76, -402.45) mm, rotated rx 0 ry 39.88 rz 90.63 deg; joints [17.695, -86.747, 125.35, -79.096, 14.145, 89.861]
  MoveL 209 to (-426.66, 202.68, -394.68) mm, rotated rx 0 ry 41.19 rz 90.37 deg; joints [17.543, -86.773, 124.541, -70.479, 14.182, 81.404]
  MoveL 210 to (-426.66, 192.61, -385.66) mm, rotated rx 0 ry 42.56 rz 90.06 deg; joints [17.368, -86.759, 123.638, -61.579, 14.521, 72.697]
  MoveL 211 to (-426.66, 181.56, -375.24) mm, rotated rx 0 ry 44.02 rz 89.7 deg; joints [17.171, -86.693, 122.626, -52.729, 15.213, 64.063]
  MoveL 212 to (-426.66, 169.68, -363.45) mm, rotated rx 0 ry 45.57 rz 89.32 deg; joints [16.955, -86.564, 121.505, -44.364, 16.286, 55.926]
  MoveL 213 to (-426.66, 157.13, -350.27) mm, rotated rx 0 ry 47.22 rz 88.95 deg; joints [16.723, -86.36, 120.269, -36.792, 17.745, 48.579]
  MoveL 214 to (-426.66, 144.06, -335.7) mm, rotated rx 0 ry 48.99 rz 88.6 deg; joints [16.478, -86.069, 118.913, -30.169, 19.577, 42.17]
  MoveL 215 to (-426.66, 130.64, -319.75) mm, rotated rx 0 ry 50.86 rz 88.28 deg; joints [16.223, -85.684, 117.44, -24.569, 21.735, 36.763]
  MoveL 216 to (-426.66, 117.01, -302.4) mm, rotated rx 0 ry 52.84 rz 88.01 deg; joints [15.962, -85.193, 115.848, -19.909, 24.183, 32.269]
  MoveL 217 to (-426.66, 103.45, -283.84) mm, rotated rx 0 ry 54.91 rz 87.8 deg; joints [15.699, -84.597, 114.15, -16.099, 26.864, 28.595]
  MoveL 218 to (-426.66, 90.56, -264.77) mm, rotated rx 0 ry 57.01 rz 87.66 deg; joints [15.445, -83.915, 112.41, -13.089, 29.645, 25.685]
  MoveL 219 to (-426.66, 78.4, -245.27) mm, rotated rx 0 ry 59.13 rz 87.58 deg; joints [15.201, -83.153, 110.63, -10.68, 32.503, 23.348]
  MoveL 220 to (-426.66, 66.99, -225.36) mm, rotated rx 0 ry 61.28 rz 87.56 deg; joints [14.966, -82.315, 108.814, -8.739, 35.41, 21.452]
  MoveL 221 to (-426.66, 56.34, -205.04) mm, rotated rx 0 ry 63.45 rz 87.59 deg; joints [14.74, -81.404, 106.962, -7.164, 38.352, 19.9]
  MoveL 222 to (-426.66, 46.46, -184.33) mm, rotated rx 0 ry 65.62 rz 87.67 deg; joints [14.525, -80.427, 105.081, -5.887, 41.299, 18.626]
  MoveL 223 to (-426.66, 37.37, -163.24) mm, rotated rx 0 ry 67.79 rz 87.8 deg; joints [14.321, -79.388, 103.173, -4.854, 44.245, 17.574]
  MoveL 224 to (-426.66, 29.08, -141.79) mm, rotated rx 0 ry 69.99 rz 87.97 deg; joints [14.126, -78.283, 101.226, -4.005, 47.225, 16.69]
  MoveL 225 to (-426.66, 21.64, -120.06) mm, rotated rx 0 ry 72.22 rz 88.19 deg; joints [13.94, -77.117, 99.246, -3.308, 50.229, 15.945]
  MoveL 226 to (-426.66, 15.06, -98.07) mm, rotated rx 0 ry 74.49 rz 88.45 deg; joints [13.763, -75.892, 97.234, -2.738, 53.255, 15.316]
  MoveL 227 to (-426.66, 15.06, -98.07) mm, rotated rx 0 ry 74.49 rz 88.45 deg; joints [13.763, -75.892, 97.234, -2.738, 53.255, 15.316]
  MoveL 228 to (-427.52, 12.32, -87.76) mm, rotated rx 0 ry 75.54 rz 88.58 deg; joints [13.664, -75.313, 96.301, -2.505, 54.655, 15.036]
  MoveL 229 to (-430.06, 9.87, -77.65) mm, rotated rx 0 ry 76.56 rz 88.71 deg; joints [13.531, -74.756, 95.413, -2.295, 55.992, 14.743]
  MoveL 230 to (-434.22, 7.74, -68.02) mm, rotated rx 0 ry 77.49 rz 88.85 deg; joints [13.367, -74.24, 94.597, -2.111, 57.226, 14.443]
  MoveL 231 to (-439.95, 5.96, -59.18) mm, rotated rx 0 ry 78.32 rz 88.97 deg; joints [13.176, -73.784, 93.88, -1.958, 58.314, 14.14]
  MoveL 232 to (-443.39, 5.2, -55.16) mm, rotated rx 0 ry 78.68 rz 89.03 deg; joints [13.072, -73.585, 93.568, -1.894, 58.788, 13.99]
  MoveL 233 to (-447.19, 4.54, -51.48) mm, rotated rx 0 ry 79 rz 89.09 deg; joints [12.962, -73.41, 93.295, -1.839, 59.207, 13.84]
  MoveL 234 to (-451.34, 3.97, -48.2) mm, rotated rx 0 ry 79.28 rz 89.14 deg; joints [12.848, -73.263, 93.063, -1.791, 59.564, 13.692]
  MoveL 235 to (-455.82, 3.5, -45.36) mm, rotated rx 0 ry 79.49 rz 89.18 deg; joints [12.729, -73.146, 92.88, -1.753, 59.85, 13.547]
  MoveL 236 to (-460.59, 3.14, -43.04) mm, rotated rx 0 ry 79.65 rz 89.21 deg; joints [12.608, -73.065, 92.749, -1.722, 60.059, 13.405]
  MoveL 237 to (-465.6, 2.89, -41.29) mm, rotated rx 0 ry 79.75 rz 89.24 deg; joints [12.486, -73.02, 92.674, -1.7, 60.184, 13.268]
  MoveL 238 to (-470.8, 2.76, -40.16) mm, rotated rx 0 ry 79.78 rz 89.26 deg; joints [12.362, -73.015, 92.661, -1.684, 60.22, 13.136]
  MoveL 239 to (-476.11, 2.74, -39.69) mm, rotated rx 0 ry 79.74 rz 89.26 deg; joints [12.241, -73.052, 92.71, -1.675, 60.165, 13.011]
  MoveL 240 to (-481.43, 2.85, -39.9) mm, rotated rx 0 ry 79.63 rz 89.25 deg; joints [12.122, -73.129, 92.821, -1.671, 60.018, 12.895]
  MoveL 241 to (-486.68, 3.08, -40.78) mm, rotated rx 0 ry 79.45 rz 89.23 deg; joints [12.009, -73.246, 92.992, -1.673, 59.784, 12.79]
  MoveL 242 to (-491.76, 3.43, -42.29) mm, rotated rx 0 ry 79.21 rz 89.2 deg; joints [11.903, -73.397, 93.217, -1.678, 59.47, 12.695]
  MoveL 243 to (-496.62, 3.91, -44.4) mm, rotated rx 0 ry 78.92 rz 89.16 deg; joints [11.804, -73.581, 93.492, -1.687, 59.084, 12.613]
  MoveL 244 to (-501.21, 4.5, -47.03) mm, rotated rx 0 ry 78.59 rz 89.11 deg; joints [11.714, -73.792, 93.81, -1.699, 58.636, 12.543]
  MoveL 245 to (-505.48, 5.21, -50.14) mm, rotated rx 0 ry 78.21 rz 89.06 deg; joints [11.634, -74.025, 94.163, -1.714, 58.135, 12.487]
  MoveL 246 to (-509.4, 6.03, -53.67) mm, rotated rx 0 ry 77.8 rz 88.99 deg; joints [11.563, -74.277, 94.548, -1.732, 57.589, 12.444]
  MoveL 247 to (-512.95, 6.94, -57.54) mm, rotated rx 0 ry 77.37 rz 88.93 deg; joints [11.502, -74.543, 94.957, -1.754, 57.006, 12.414]
  MoveL 248 to (-518.87, 9.07, -66.17) mm, rotated rx 0 ry 76.44 rz 88.78 deg; joints [11.411, -75.106, 95.83, -1.808, 55.761, 12.397]
  MoveL 249 to (-523.17, 11.54, -75.64) mm, rotated rx 0 ry 75.47 rz 88.63 deg; joints [11.363, -75.691, 96.748, -1.88, 54.446, 12.436]
  MoveL 250 to (-525.78, 14.29, -85.65) mm, rotated rx 0 ry 74.48 rz 88.48 deg; joints [11.357, -76.278, 97.682, -1.976, 53.102, 12.536]
  MoveL 251 to (-526.66, 17.25, -95.89) mm, rotated rx 0 ry 73.5 rz 88.33 deg; joints [11.394, -76.85, 98.608, -2.1, 51.762, 12.697]
  MoveL 252 to (-526.66, 17.25, -95.89) mm, rotated rx 0 ry 73.5 rz 88.33 deg; joints [11.394, -76.85, 98.608, -2.1, 51.762, 12.697]
  MoveL 253 to (-526.66, 23.7, -116.37) mm, rotated rx 0 ry 71.57 rz 88.08 deg; joints [11.518, -77.951, 100.424, -2.421, 49.114, 13.118]
  MoveL 254 to (-526.66, 30.84, -136.65) mm, rotated rx 0 ry 69.67 rz 87.86 deg; joints [11.65, -79.005, 102.213, -2.838, 46.489, 13.619]
  MoveL 255 to (-526.66, 38.67, -156.75) mm, rotated rx 0 ry 67.8 rz 87.69 deg; joints [11.791, -80.013, 103.976, -3.366, 43.884, 14.215]
  MoveL 256 to (-526.66, 47.17, -176.64) mm, rotated rx 0 ry 65.95 rz 87.56 deg; joints [11.942, -80.971, 105.712, -4.028, 41.301, 14.923]
  MoveL 257 to (-526.66, 56.34, -196.3) mm, rotated rx 0 ry 64.12 rz 87.49 deg; joints [12.102, -81.882, 107.425, -4.854, 38.729, 15.774]
  MoveL 258 to (-526.66, 66.15, -215.69) mm, rotated rx 0 ry 62.25 rz 87.46 deg; joints [12.273, -82.75, 109.132, -5.905, 36.104, 16.823]
  MoveL 259 to (-526.66, 76.6, -234.78) mm, rotated rx 0 ry 60.4 rz 87.48 deg; joints [12.454, -83.562, 110.811, -7.197, 33.5, 18.09]
  MoveL 260 to (-526.66, 87.66, -253.52) mm, rotated rx 0 ry 58.56 rz 87.55 deg; joints [12.644, -84.315, 112.461, -8.791, 30.919, 19.633]
  MoveL 261 to (-526.66, 99.1, -271.59) mm, rotated rx 0 ry 56.8 rz 87.67 deg; joints [12.839, -84.992, 114.045, -10.711, 28.436, 21.476]
  MoveL 262 to (-526.66, 110.75, -288.81) mm, rotated rx 0 ry 55.1 rz 87.84 deg; joints [13.037, -85.592, 115.557, -13.016, 26.067, 23.679]
  MoveL 263 to (-526.66, 122.53, -305.17) mm, rotated rx 0 ry 53.46 rz 88.06 deg; joints [13.237, -86.116, 116.998, -15.79, 23.811, 26.324]
  MoveL 264 to (-526.66, 134.33, -320.63) mm, rotated rx 0 ry 51.87 rz 88.32 deg; joints [13.437, -86.567, 118.368, -19.126, 21.677, 29.511]
  MoveL 265 to (-526.66, 146.06, -335.17) mm, rotated rx 0 ry 50.32 rz 88.61 deg; joints [13.636, -86.948, 119.67, -23.145, 19.672, 33.363]
  MoveL 266 to (-526.66, 157.63, -348.74) mm, rotated rx 0 ry 48.79 rz 88.91 deg; joints [13.83, -87.264, 120.907, -28.004, 17.802, 38.044]
  MoveL 267 to (-526.66, 168.94, -361.33) mm, rotated rx 0 ry 47.28 rz 89.21 deg; joints [14.018, -87.515, 122.078, -33.857, 16.094, 43.72]
  MoveL 268 to (-526.66, 179.9, -372.89) mm, rotated rx 0 ry 45.77 rz 89.48 deg; joints [14.195, -87.706, 123.191, -40.945, 14.562, 50.644]
  MoveL 269 to (-526.66, 190.36, -383.36) mm, rotated rx 0 ry 44.21 rz 89.7 deg; joints [14.358, -87.84, 124.251, -49.587, 13.232, 59.149]
  MoveL 270 to (-526.66, 200.13, -392.6) mm, rotated rx 0 ry 42.59 rz 89.85 deg; joints [14.503, -87.92, 125.254, -59.973, 12.178, 69.443]
  MoveL 271 to (-526.66, 209.21, -400.7) mm, rotated rx 0 ry 40.89 rz 89.89 deg; joints [14.629, -87.946, 126.209, -72.219, 11.493, 81.655]
  MoveL 272 to (-526.66, 217.6, -407.74) mm, rotated rx 0 ry 39.1 rz 89.82 deg; joints [14.736, -87.921, 127.123, -85.906, 11.305, 95.377]
  MoveL 273 to (-526.66, 225.31, -413.8) mm, rotated rx 0 ry 37.22 rz 89.64 deg; joints [14.823, -87.841, 127.994, -99.845, 11.714, 109.426]
  MoveL 274 to (-526.66, 232.35, -418.97) mm, rotated rx 0 ry 35.3 rz 89.34 deg; joints [14.892, -87.709, 128.816, -112.541, 12.717, 122.311]
  MoveL 275 to (-526.66, 238.74, -423.35) mm, rotated rx 0 ry 33.38 rz 88.94 deg; joints [14.946, -87.529, 129.577, -123.033, 14.194, 133.068]
  MoveL 276 to (-526.66, 244.48, -427) mm, rotated rx 0 ry 31.53 rz 88.47 deg; joints [14.985, -87.308, 130.264, -131.171, 15.957, 141.533]
  MoveL 277 to (-526.66, 249.59, -430.03) mm, rotated rx 0 ry 29.8 rz 87.96 deg; joints [15.014, -87.061, 130.869, -137.281, 17.824, 148.017]
  MoveL 278 to (-526.66, 254.07, -432.51) mm, rotated rx 0 ry 28.25 rz 87.42 deg; joints [15.034, -86.803, 131.391, -141.818, 19.654, 152.954]
  MoveL 279 to (-526.66, 262.06, -436.56) mm, rotated rx 0 ry 25.44 rz 86.27 deg; joints [15.059, -86.249, 132.276, -148.219, 23.219, 160.252]
  MoveL 280 to (-526.66, 268.98, -439.66) mm, rotated rx 0 ry 22.87 rz 84.89 deg; joints [15.065, -85.65, 133.017, -152.689, 26.684, 165.848]
  MoveL 281 to (-526.66, 274.79, -441.94) mm, rotated rx 0 ry 20.27 rz 82.87 deg; joints [15.038, -84.985, 133.68, -156.396, 30.274, 171.243]
  MoveL 282 to (-526.66, 274.79, -441.94) mm, rotated rx 0 ry 20.27 rz 82.87 deg; joints [15.038, -84.985, 133.68, -156.396, 30.274, 171.243]
  MoveL 283 to (-528.26, 284.84, -445.08) mm, rotated rx 0 ry 15.98 rz 77.87 deg; joints [14.91, -83.662, 134.682, -161.262, 36.583, 180.489]
  MoveL 284 to (-531.46, 294.75, -447.3) mm, rotated rx 0 ry 12.61 rz 71.28 deg; joints [14.726, -82.329, 135.412, -164.374, 42.016, 189.626]
  MoveL 285 to (-536.1, 304.3, -448.73) mm, rotated rx 0 ry 10.33 rz 63.96 deg; joints [14.509, -81.16, 135.907, -166.347, 46.155, 198.478]
  MoveL 286 to (-542.07, 313.14, -449.53) mm, rotated rx 0 ry 8.92 rz 56.9 deg; joints [14.265, -80.21, 136.246, -167.678, 49.135, 206.509]
  MoveL 287 to (-549.34, 320.94, -449.83) mm, rotated rx 0 ry 8.08 rz 50.8 deg; joints [13.989, -79.467, 136.489, -168.673, 51.248, 213.307]
  MoveL 288 to (-553.45, 324.34, -449.81) mm, rotated rx 0 ry 7.8 rz 48.22 deg; joints [13.838, -79.168, 136.586, -169.098, 52.049, 216.171]
  MoveL 289 to (-557.86, 327.32, -449.7) mm, rotated rx 0 ry 7.6 rz 45.98 deg; joints [13.678, -78.918, 136.67, -169.492, 52.704, 218.66]
  MoveL 290 to (-562.55, 329.81, -449.5) mm, rotated rx 0 ry 7.46 rz 44.1 deg; joints [13.51, -78.717, 136.744, -169.863, 53.224, 220.772]
  MoveL 291 to (-567.49, 331.76, -449.2) mm, rotated rx 0 ry 7.37 rz 42.58 deg; joints [13.333, -78.567, 136.807, -170.214, 53.618, 222.509]
  MoveL 292 to (-572.6, 333.08, -448.83) mm, rotated rx 0 ry 7.32 rz 41.41 deg; joints [13.151, -78.471, 136.861, -170.548, 53.888, 223.863]
  MoveL 293 to (-577.85, 333.73, -448.38) mm, rotated rx 0 ry 7.3 rz 40.61 deg; joints [12.965, -78.43, 136.904, -170.865, 54.036, 224.841]
  MoveL 294 to (-583.14, 333.65, -447.85) mm, rotated rx 0 ry 7.32 rz 40.17 deg; joints [12.778, -78.446, 136.937, -171.162, 54.064, 225.442]
  MoveL 295 to (-588.37, 332.84, -447.27) mm, rotated rx 0 ry 7.37 rz 40.08 deg; joints [12.594, -78.519, 136.959, -171.437, 53.971, 225.666]
  MoveL 296 to (-593.42, 331.32, -446.64) mm, rotated rx 0 ry 7.45 rz 40.35 deg; joints [12.415, -78.647, 136.969, -171.685, 53.761, 225.521]
  MoveL 297 to (-598.22, 329.15, -445.97) mm, rotated rx 0 ry 7.56 rz 40.95 deg; joints [12.247, -78.827, 136.968, -171.901, 53.437, 225.017]
  MoveL 298 to (-602.71, 326.38, -445.28) mm, rotated rx 0 ry 7.7 rz 41.88 deg; joints [12.09, -79.054, 136.955, -172.083, 53.001, 224.162]
  MoveL 299 to (-606.82, 323.1, -444.56) mm, rotated rx 0 ry 7.87 rz 43.13 deg; joints [11.947, -79.324, 136.929, -172.226, 52.457, 222.97]
  MoveL 300 to (-610.56, 319.39, -443.82) mm, rotated rx 0 ry 8.08 rz 44.68 deg; joints [11.818, -79.633, 136.89, -172.328, 51.801, 221.444]
  MoveL 301 to (-613.91, 315.31, -443.06) mm, rotated rx 0 ry 8.34 rz 46.54 deg; joints [11.705, -79.98, 136.837, -172.384, 51.029, 219.585]
  MoveL 302 to (-619.41, 306.3, -441.48) mm, rotated rx 0 ry 9.03 rz 51.15 deg; joints [11.525, -80.779, 136.682, -172.336, 49.097, 214.883]
  MoveL 303 to (-623.33, 296.51, -439.76) mm, rotated rx 0 ry 10.08 rz 56.83 deg; joints [11.412, -81.718, 136.445, -172.008, 46.535, 208.921]
  MoveL 304 to (-625.71, 286.27, -437.84) mm, rotated rx 0 ry 11.69 rz 63.35 deg; joints [11.369, -82.807, 136.088, -171.256, 43.124, 201.836]
  MoveL 305 to (-626.52, 275.84, -435.58) mm, rotated rx 0 ry 14.15 rz 70.2 deg; joints [11.403, -84.056, 135.544, -169.786, 38.549, 193.858]
  MoveL 306 to (-626.52, 275.84, -435.58) mm, rotated rx 0 ry 14.15 rz 70.2 deg; joints [11.403, -84.056, 135.544, -169.786, 38.549, 193.858]
  MoveL 307 to (-626.52, 264.53, -432.46) mm, rotated rx 0 ry 18.11 rz 77.07 deg; joints [11.499, -85.535, 134.638, -166.775, 32.017, 184.538]
  MoveL 308 to (-626.52, 254.35, -428.73) mm, rotated rx 0 ry 22.84 rz 82.03 deg; joints [11.595, -86.824, 133.458, -161.675, 24.93, 175.109]
  MoveL 309 to (-626.52, 244.87, -424.28) mm, rotated rx 0 ry 27.72 rz 85.28 deg; joints [11.663, -87.777, 132.094, -153.158, 18.255, 163.951]
  MoveL 310 to (-626.52, 235.54, -418.96) mm, rotated rx 0 ry 31.51 rz 86.81 deg; joints [11.657, -88.333, 130.847, -141.936, 13.481, 151.553]
  MoveL 311 to (-626.52, 226.61, -413.13) mm, rotated rx 0 ry 34.69 rz 87.7 deg; joints [11.621, -88.658, 129.678, -125.609, 10.149, 134.577]
  MoveL 312 to (-626.52, 218.14, -406.95) mm, rotated rx 0 ry 37.51 rz 88.33 deg; joints [11.571, -88.829, 128.548, -102.244, 8.338, 110.783]
  MoveL 313 to (-626.52, 209.6, -400.09) mm, rotated rx 0 ry 40.08 rz 88.76 deg; joints [11.506, -88.887, 127.425, -76.013, 8.236, 84.271]
  MoveL 314 to (-626.52, 200.94, -392.5) mm, rotated rx 0 ry 42.37 rz 89.03 deg; joints [11.426, -88.855, 126.322, -55.471, 9.442, 63.568]
  MoveL 315 to (-626.52, 192.12, -384.14) mm, rotated rx 0 ry 44.4 rz 89.15 deg; joints [11.332, -88.753, 125.242, -41.99, 11.224, 50.018]
  MoveL 316 to (-626.52, 183.07, -374.99) mm, rotated rx 0 ry 46.2 rz 89.16 deg; joints [11.225, -88.595, 124.177, -33.108, 13.155, 41.138]
  MoveL 317 to (-626.52, 173.72, -364.95) mm, rotated rx 0 ry 47.82 rz 89.07 deg; joints [11.105, -88.388, 123.111, -26.842, 15.09, 34.927]
  MoveL 318 to (-626.52, 164.06, -354.01) mm, rotated rx 0 ry 49.3 rz 88.92 deg; joints [10.975, -88.135, 122.031, -22.131, 16.991, 30.308]
  MoveL 319 to (-626.52, 154.16, -342.2) mm, rotated rx 0 ry 50.73 rz 88.72 deg; joints [10.836, -87.834, 120.92, -18.369, 18.893, 26.662]
  MoveL 320 to (-626.52, 144.09, -329.59) mm, rotated rx 0 ry 52.08 rz 88.5 deg; joints [10.692, -87.489, 119.781, -15.323, 20.772, 23.744]
  MoveL 321 to (-626.52, 133.91, -316.21) mm, rotated rx 0 ry 53.41 rz 88.27 deg; joints [10.545, -87.097, 118.608, -12.8, 22.653, 21.349]
  MoveL 322 to (-626.52, 123.68, -302.1) mm, rotated rx 0 ry 54.72 rz 88.06 deg; joints [10.398, -86.657, 117.395, -10.682, 24.556, 19.353]
  MoveL 323 to (-626.52, 113.48, -287.33) mm, rotated rx 0 ry 56.05 rz 87.86 deg; joints [10.251, -86.168, 116.14, -8.895, 26.495, 17.674]
  MoveL 324 to (-626.52, 103.37, -271.93) mm, rotated rx 0 ry 57.39 rz 87.7 deg; joints [10.107, -85.628, 114.84, -7.385, 28.479, 16.255]
  MoveL 325 to (-626.52, 93.42, -255.97) mm, rotated rx 0 ry 58.77 rz 87.57 deg; joints [9.967, -85.039, 113.496, -6.111, 30.512, 15.052]
  MoveL 326 to (-626.52, 84.08, -240.14) mm, rotated rx 0 ry 60.15 rz 87.48 deg; joints [9.837, -84.421, 112.156, -5.066, 32.538, 14.056]
  MoveL 327 to (-626.52, 75.49, -224.77) mm, rotated rx 0 ry 61.49 rz 87.43 deg; joints [9.717, -83.795, 110.857, -4.234, 34.483, 13.253]
  MoveL 328 to (-626.52, 67.62, -209.91) mm, rotated rx 0 ry 62.77 rz 87.42 deg; joints [9.609, -83.167, 109.6, -3.569, 36.35, 12.597]
  MoveL 329 to (-626.52, 60.45, -195.63) mm, rotated rx 0 ry 64 rz 87.43 deg; joints [9.512, -82.542, 108.39, -3.035, 38.135, 12.06]
  MoveL 330 to (-626.52, 53.95, -181.99) mm, rotated rx 0 ry 65.12 rz 87.47 deg; joints [9.425, -81.938, 107.25, -2.629, 39.77, 11.634]
  MoveL 331 to (-626.52, 48.09, -169.05) mm, rotated rx 0 ry 66.17 rz 87.52 deg; joints [9.349, -81.352, 106.171, -2.313, 41.302, 11.287]
  MoveL 332 to (-626.52, 42.84, -156.88) mm, rotated rx 0 ry 67.17 rz 87.6 deg; joints [9.281, -80.787, 105.151, -2.066, 42.746, 11]
  MoveL 333 to (-626.52, 38.17, -145.54) mm, rotated rx 0 ry 68.11 rz 87.69 deg; joints [9.222, -80.248, 104.197, -1.875, 44.093, 10.763]
  MoveL 334 to (-626.52, 34.04, -135.05) mm, rotated rx 0 ry 68.98 rz 87.78 deg; joints [9.17, -79.741, 103.312, -1.728, 45.34, 10.568]
  MoveL 335 to (-626.52, 26.46, -114.43) mm, rotated rx 0 ry 70.7 rz 88 deg; joints [9.075, -78.717, 101.563, -1.515, 47.793, 10.241]
  MoveL 336 to (-626.52, 19.52, -93.61) mm, rotated rx 0 ry 72.45 rz 88.27 deg; joints [8.989, -77.649, 99.785, -1.387, 50.273, 9.978]
  MoveL 337 to (-626.52, 19.52, -93.61) mm, rotated rx 0 ry 72.45 rz 88.27 deg; joints [8.989, -77.649, 99.785, -1.387, 50.273, 9.978]
  MoveL 338 to (-627.39, 16.45, -83.57) mm, rotated rx 0 ry 73.29 rz 88.41 deg; joints [8.93, -77.13, 98.934, -1.347, 51.455, 9.848]
  MoveL 339 to (-629.96, 13.64, -73.73) mm, rotated rx 0 ry 74.09 rz 88.56 deg; joints [8.834, -76.629, 98.122, -1.316, 52.578, 9.688]
  MoveL 340 to (-634.17, 11.15, -64.4) mm, rotated rx 0 ry 74.82 rz 88.71 deg; joints [8.703, -76.165, 97.375, -1.295, 53.602, 9.504]
  MoveL 341 to (-639.97, 9.01, -55.88) mm, rotated rx 0 ry 75.45 rz 88.86 deg; joints [8.541, -75.757, 96.719, -1.283, 54.488, 9.298]
  MoveL 342 to (-643.43, 8.09, -52.03) mm, rotated rx 0 ry 75.72 rz 88.92 deg; joints [8.448, -75.579, 96.435, -1.279, 54.866, 9.188]
  MoveL 343 to (-647.26, 7.27, -48.53) mm, rotated rx 0 ry 75.95 rz 88.99 deg; joints [8.349, -75.423, 96.185, -1.277, 55.194, 9.074]
  MoveL 344 to (-651.43, 6.57, -45.41) mm, rotated rx 0 ry 76.13 rz 89.04 deg; joints [8.244, -75.292, 95.974, -1.275, 55.466, 8.955]
  MoveL 345 to (-655.9, 5.98, -42.74) mm, rotated rx 0 ry 76.28 rz 89.09 deg; joints [8.133, -75.188, 95.807, -1.272, 55.675, 8.833]
  MoveL 346 to (-660.63, 5.53, -40.56) mm, rotated rx 0 ry 76.37 rz 89.13 deg; joints [8.017, -75.114, 95.686, -1.268, 55.819, 8.708]
  MoveL 347 to (-665.61, 5.21, -38.93) mm, rotated rx 0 ry 76.41 rz 89.16 deg; joints [7.898, -75.071, 95.614, -1.261, 55.892, 8.58]
  MoveL 348 to (-670.75, 5.03, -37.87) mm, rotated rx 0 ry 76.4 rz 89.18 deg; joints [7.775, -75.062, 95.596, -1.25, 55.892, 8.45]
  MoveL 349 to (-675.98, 4.99, -37.44) mm, rotated rx 0 ry 76.34 rz 89.19 deg; joints [7.652, -75.087, 95.631, -1.234, 55.819, 8.32]
  MoveL 350 to (-681.23, 5.11, -37.63) mm, rotated rx 0 ry 76.23 rz 89.18 deg; joints [7.53, -75.146, 95.719, -1.212, 55.673, 8.191]
  MoveL 351 to (-686.41, 5.39, -38.43) mm, rotated rx 0 ry 76.06 rz 89.17 deg; joints [7.41, -75.238, 95.859, -1.185, 55.459, 8.065]
  MoveL 352 to (-691.45, 5.81, -39.84) mm, rotated rx 0 ry 75.86 rz 89.14 deg; joints [7.294, -75.359, 96.046, -1.152, 55.183, 7.942]
  MoveL 353 to (-696.28, 6.39, -41.8) mm, rotated rx 0 ry 75.61 rz 89.09 deg; joints [7.183, -75.508, 96.276, -1.113, 54.85, 7.824]
  MoveL 354 to (-700.86, 7.1, -44.26) mm, rotated rx 0 ry 75.34 rz 89.04 deg; joints [7.079, -75.68, 96.545, -1.07, 54.469, 7.712]
  MoveL 355 to (-705.13, 7.95, -47.2) mm, rotated rx 0 ry 75.03 rz 88.99 deg; joints [6.983, -75.872, 96.848, -1.023, 54.047, 7.607]
  MoveL 356 to (-709.07, 8.93, -50.54) mm, rotated rx 0 ry 74.7 rz 88.92 deg; joints [6.894, -76.081, 97.179, -0.972, 53.59, 7.511]
  MoveL 357 to (-712.65, 10.02, -54.23) mm, rotated rx 0 ry 74.36 rz 88.85 deg; joints [6.815, -76.304, 97.533, -0.92, 53.106, 7.423]
  MoveL 358 to (-718.64, 12.52, -62.5) mm, rotated rx 0 ry 73.63 rz 88.7 deg; joints [6.684, -76.78, 98.296, -0.814, 52.075, 7.279]
  MoveL 359 to (-722.99, 15.38, -71.65) mm, rotated rx 0 ry 72.87 rz 88.54 deg; joints [6.594, -77.279, 99.106, -0.716, 50.994, 7.18]
  MoveL 360 to (-725.63, 18.51, -81.35) mm, rotated rx 0 ry 72.11 rz 88.39 deg; joints [6.548, -77.786, 99.938, -0.633, 49.895, 7.133]
  MoveL 361 to (-726.52, 21.83, -91.31) mm, rotated rx 0 ry 71.36 rz 88.24 deg; joints [6.545, -78.286, 100.766, -0.575, 48.807, 7.141]
  MoveL 362 to (-726.52, 21.83, -91.31) mm, rotated rx 0 ry 71.36 rz 88.24 deg; joints [6.545, -78.286, 100.766, -0.575, 48.807, 7.141]
  MoveL 363 to (-726.52, 32.85, -121.97) mm, rotated rx 0 ry 69.12 rz 87.86 deg; joints [6.619, -79.763, 103.268, -0.521, 45.515, 7.309]
  MoveL 364 to (-726.52, 45.08, -152.25) mm, rotated rx 0 ry 66.95 rz 87.6 deg; joints [6.714, -81.157, 105.711, -0.644, 42.283, 7.59]
  MoveL 365 to (-726.52, 58.45, -182.11) mm, rotated rx 0 ry 64.86 rz 87.47 deg; joints [6.83, -82.464, 108.093, -0.979, 39.121, 8.016]
  MoveL 366 to (-726.52, 72.8, -211.24) mm, rotated rx 0 ry 62.72 rz 87.45 deg; joints [6.969, -83.695, 110.441, -1.603, 35.889, 8.657]
  MoveL 367 to (-726.52, 88.21, -239.78) mm, rotated rx 0 ry 60.55 rz 87.55 deg; joints [7.13, -84.845, 112.757, -2.561, 32.603, 9.568]
  MoveL 368 to (-726.52, 104.86, -267.98) mm, rotated rx 0 ry 58.39 rz 87.76 deg; joints [7.312, -85.91, 115.049, -3.942, 29.285, 10.841]
  MoveL 369 to (-726.52, 113.8, -282.17) mm, rotated rx 0 ry 57.28 rz 87.9 deg; joints [7.412, -86.415, 116.204, -4.849, 27.586, 11.67]
  MoveL 370 to (-726.52, 123.24, -296.54) mm, rotated rx 0 ry 56.12 rz 88.07 deg; joints [7.519, -86.91, 117.389, -5.965, 25.8, 12.693]
  MoveL 371 to (-726.52, 143.33, -325.06) mm, rotated rx 0 ry 53.51 rz 88.44 deg; joints [7.749, -87.841, 119.831, -9.044, 21.872, 15.561]
  MoveL 372 to (-726.52, 153.81, -338.84) mm, rotated rx 0 ry 51.98 rz 88.61 deg; joints [7.866, -88.268, 121.097, -11.217, 19.63, 17.639]
  MoveL 373 to (-726.52, 164.46, -352.04) mm, rotated rx 0 ry 50.19 rz 88.71 deg; joints [7.979, -88.663, 122.407, -14.138, 17.094, 20.497]
  MoveL 374 to (-726.52, 175.2, -364.47) mm, rotated rx 0 ry 48.1 rz 88.72 deg; joints [8.082, -89.011, 123.766, -18.373, 14.216, 24.726]
  MoveL 375 to (-726.52, 185.95, -375.96) mm, rotated rx 0 ry 45.58 rz 88.57 deg; joints [8.17, -89.295, 125.191, -25.594, 10.915, 32.035]
  MoveL 376 to (-726.52, 191.23, -381.21) mm, rotated rx 0 ry 44.17 rz 88.42 deg; joints [8.206, -89.402, 125.918, -31.578, 9.166, 38.107]
  MoveL 377 to (-726.52, 196.27, -385.97) mm, rotated rx 0 ry 42.7 rz 88.23 deg; joints [8.237, -89.477, 126.629, -40.438, 7.494, 47.088]
  MoveL 378 to (-726.52, 201.05, -390.27) mm, rotated rx 0 ry 41.21 rz 88 deg; joints [8.261, -89.519, 127.314, -54.003, 6.057, 60.804]
  MoveL 379 to (-726.52, 205.55, -394.11) mm, rotated rx 0 ry 39.72 rz 87.73 deg; joints [8.28, -89.529, 127.967, -73.949, 5.121, 80.928]
  MoveL 380 to (-726.52, 209.74, -397.51) mm, rotated rx 0 ry 38.26 rz 87.44 deg; joints [8.295, -89.508, 128.578, -97.902, 4.975, 105.083]
  MoveL 381 to (-726.52, 213.61, -400.49) mm, rotated rx 0 ry 36.87 rz 87.13 deg; joints [8.305, -89.46, 129.139, -118.696, 5.614, 126.097]
  MoveL 382 to (-726.52, 217.13, -403.06) mm, rotated rx 0 ry 35.58 rz 86.81 deg; joints [8.313, -89.391, 129.645, -132.967, 6.714, 140.597]
  MoveL 383 to (-726.52, 220.28, -405.25) mm, rotated rx 0 ry 34.15 rz 86.34 deg; joints [8.306, -89.295, 130.157, -143.949, 8.213, 151.924]
  MoveL 384 to (-726.52, 225.45, -408.57) mm, rotated rx 0 ry 31.24 rz 85.07 deg; joints [8.264, -89.032, 131.108, -157.251, 11.75, 166.18]
  MoveL 385 to (-726.52, 230.33, -411.35) mm, rotated rx 0 ry 28.36 rz 83.5 deg; joints [8.209, -88.667, 131.985, -164.398, 15.62, 174.553]
  MoveL 386 to (-726.52, 240.81, -416.26) mm, rotated rx 0 ry 22.49 rz 78.97 deg; joints [8.071, -87.557, 133.624, -171.968, 24.183, 185.911]
  MoveL 387 to (-726.52, 252.74, -420.41) mm, rotated rx 0 ry 17.28 rz 72.25 deg; joints [7.929, -86.044, 134.938, -175.518, 32.527, 195.466]
  MoveL 388 to (-726.52, 259.42, -422.23) mm, rotated rx 0 ry 15.13 rz 68.03 deg; joints [7.867, -85.206, 135.454, -176.571, 36.28, 200.421]
  MoveL 389 to (-726.52, 266.67, -423.91) mm, rotated rx 0 ry 13.33 rz 63.31 deg; joints [7.814, -84.348, 135.884, -177.334, 39.676, 205.63]
  MoveL 390 to (-726.52, 266.67, -423.91) mm, rotated rx 0 ry 13.33 rz 63.31 deg; joints [7.814, -84.348, 135.884, -177.334, 39.676, 205.63]
  MoveL 391 to (-727.38, 277.72, -425.89) mm, rotated rx 0 ry 11.38 rz 56.11 deg; joints [7.725, -83.154, 136.364, -178.117, 43.795, 213.275]
  MoveL 392 to (-729.84, 288.66, -427.25) mm, rotated rx 0 ry 10.12 rz 49.34 deg; joints [7.6, -82.093, 136.704, -178.693, 46.952, 220.337]
  MoveL 393 to (-733.81, 299.23, -428.09) mm, rotated rx 0 ry 9.33 rz 43.46 deg; joints [7.435, -81.165, 136.949, -179.174, 49.382, 226.457]
  MoveL 394 to (-739.2, 309.14, -428.48) mm, rotated rx 0 ry 8.85 rz 38.6 deg; joints [7.229, -80.359, 137.13, -179.623, 51.266, 231.522]
  MoveL 395 to (-746.01, 318.12, -428.47) mm, rotated rx 0 ry 8.55 rz 34.75 deg; joints [6.978, -79.668, 137.263, -180.081, 52.734, 235.598]
  MoveL 396 to (-749.94, 322.15, -428.31) mm, rotated rx 0 ry 8.46 rz 33.17 deg; joints [6.836, -79.368, 137.315, -180.321, 53.334, 237.291]
  MoveL 397 to (-754.21, 325.79, -428.07) mm, rotated rx 0 ry 8.39 rz 31.8 deg; joints [6.681, -79.1, 137.358, -180.57, 53.85, 238.773]
  MoveL 398 to (-758.83, 328.97, -427.73) mm, rotated rx 0 ry 8.34 rz 30.65 deg; joints [6.515, -78.868, 137.392, -180.83, 54.284, 240.051]
  MoveL 399 to (-763.75, 331.63, -427.3) mm, rotated rx 0 ry 8.32 rz 29.7 deg; joints [6.339, -78.675, 137.418, -181.102, 54.636, 241.133]
  MoveL 400 to (-768.94, 333.68, -426.79) mm, rotated rx 0 ry 8.31 rz 28.95 deg; joints [6.153, -78.527, 137.435, -181.384, 54.902, 242.021]
  MoveL 401 to (-774.34, 335.02, -426.19) mm, rotated rx 0 ry 8.33 rz 28.4 deg; joints [5.96, -78.426, 137.443, -181.674, 55.078, 242.715]
  MoveL 402 to (-779.87, 335.61, -425.52) mm, rotated rx 0 ry 8.35 rz 28.05 deg; joints [5.762, -78.378, 137.443, -181.971, 55.161, 243.214]
  MoveL 403 to (-785.42, 335.37, -424.78) mm, rotated rx 0 ry 8.39 rz 27.91 deg; joints [5.564, -78.385, 137.433, -182.268, 55.149, 243.515]
  MoveL 404 to (-790.87, 334.32, -423.99) mm, rotated rx 0 ry 8.45 rz 27.97 deg; joints [5.37, -78.448, 137.414, -182.561, 55.04, 243.616]
  MoveL 405 to (-796.09, 332.47, -423.18) mm, rotated rx 0 ry 8.51 rz 28.22 deg; joints [5.184, -78.564, 137.387, -182.844, 54.838, 243.519]
  MoveL 406 to (-800.98, 329.9, -422.35) mm, rotated rx 0 ry 8.59 rz 28.67 deg; joints [5.009, -78.73, 137.351, -183.112, 54.547, 243.226]
  MoveL 407 to (-805.49, 326.69, -421.51) mm, rotated rx 0 ry 8.68 rz 29.31 deg; joints [4.849, -78.941, 137.308, -183.363, 54.173, 242.741]
  MoveL 408 to (-809.57, 322.95, -420.68) mm, rotated rx 0 ry 8.78 rz 30.13 deg; joints [4.705, -79.19, 137.258, -183.592, 53.722, 242.067]
  MoveL 409 to (-813.21, 318.76, -419.86) mm, rotated rx 0 ry 8.89 rz 31.14 deg; joints [4.577, -79.473, 137.2, -183.8, 53.195, 241.202]
  MoveL 410 to (-816.39, 314.19, -419.06) mm, rotated rx 0 ry 9.02 rz 32.34 deg; joints [4.466, -79.787, 137.135, -183.985, 52.595, 240.141]
  MoveL 411 to (-819.12, 309.33, -418.27) mm, rotated rx 0 ry 9.17 rz 33.73 deg; joints [4.372, -80.127, 137.063, -184.146, 51.923, 238.88]
  MoveL 412 to (-823.26, 298.97, -416.72) mm, rotated rx 0 ry 9.54 rz 37.13 deg; joints [4.234, -80.877, 136.895, -184.395, 50.348, 235.724]
  MoveL 413 to (-825.71, 288.07, -415.21) mm, rotated rx 0 ry 10.06 rz 41.41 deg; joints [4.162, -81.713, 136.688, -184.538, 48.419, 231.649]
  MoveL 414 to (-826.52, 276.9, -413.68) mm, rotated rx 0 ry 10.81 rz 46.66 deg; joints [4.157, -82.637, 136.428, -184.558, 46.027, 226.569]
  MoveL 415 to (-826.52, 276.9, -413.68) mm, rotated rx 0 ry 10.81 rz 46.66 deg; joints [4.157, -82.637, 136.428, -184.558, 46.027, 226.569]
  MoveL 416 to (-826.52, 269.11, -412.52) mm, rotated rx 0 ry 11.54 rz 50.83 deg; joints [4.182, -83.334, 136.204, -184.507, 44.018, 222.492]
  MoveL 417 to (-826.52, 261.9, -411.3) mm, rotated rx 0 ry 12.44 rz 55.01 deg; joints [4.212, -84.023, 135.95, -184.425, 41.833, 218.401]
  MoveL 418 to (-826.52, 249, -408.64) mm, rotated rx 0 ry 14.81 rz 63.05 deg; joints [4.293, -85.388, 135.328, -184.129, 36.829, 210.472]
  MoveL 419 to (-826.52, 237.74, -405.61) mm, rotated rx 0 ry 18.08 rz 70.19 deg; joints [4.404, -86.717, 134.5, -183.562, 30.849, 203.258]
  MoveL 420 to (-826.52, 227.87, -402.16) mm, rotated rx 0 ry 22.25 rz 76.04 deg; joints [4.544, -87.928, 133.417, -182.5, 23.947, 196.913]
  MoveL 421 to (-826.52, 219.11, -398.23) mm, rotated rx 0 ry 27.11 rz 80.53 deg; joints [4.7, -88.9, 132.073, -180.353, 16.466, 190.898]
  MoveL 422 to (-826.52, 211.2, -393.77) mm, rotated rx 0 ry 32.21 rz 83.78 deg; joints [4.853, -89.537, 130.54, -174.887, 9.041, 182.797]
  MoveL 423 to (-826.52, 203.64, -388.56) mm, rotated rx 0 ry 37.15 rz 86.03 deg; joints [4.981, -89.835, 128.909, -141.772, 2.556, 147.964]
  MoveL 424 to (-826.52, 199.57, -385.33) mm, rotated rx 0 ry 39.6 rz 86.9 deg; joints [5.032, -89.873, 128.037, -53.919, 2.361, 59.486]
  MoveL 425 to (-826.52, 195.07, -381.46) mm, rotated rx 0 ry 41.65 rz 87.44 deg; joints [5.053, -89.85, 127.221, -26.016, 4.736, 31.21]
  MoveL 426 to (-826.52, 189.97, -376.78) mm, rotated rx 0 ry 43.43 rz 87.74 deg; joints [5.049, -89.781, 126.426, -17.389, 7.103, 22.372]
  MoveL 427 to (-826.52, 184.24, -371.18) mm, rotated rx 0 ry 45.31 rz 88.02 deg; joints [5.04, -89.659, 125.54, -12.838, 9.669, 17.637]
  MoveL 428 to (-826.52, 177.86, -364.51) mm, rotated rx 0 ry 47.22 rz 88.25 deg; joints [5.022, -89.476, 124.576, -10.024, 12.315, 14.673]
  MoveL 429 to (-826.52, 170.81, -356.62) mm, rotated rx 0 ry 49.1 rz 88.42 deg; joints [4.994, -89.23, 123.543, -8.063, 14.95, 12.606]
  MoveL 430 to (-826.52, 163.07, -347.38) mm, rotated rx 0 ry 50.94 rz 88.51 deg; joints [4.954, -88.921, 122.444, -6.535, 17.54, 11.019]
  MoveL 431 to (-826.52, 154.62, -336.64) mm, rotated rx 0 ry 52.66 rz 88.53 deg; joints [4.9, -88.55, 121.29, -5.268, 20.013, 9.742]
  MoveL 432 to (-826.52, 145.44, -324.25) mm, rotated rx 0 ry 54.26 rz 88.47 deg; joints [4.834, -88.12, 120.081, -4.159, 22.349, 8.667]
  MoveL 433 to (-826.52, 140.57, -317.4) mm, rotated rx 0 ry 55.01 rz 88.41 deg; joints [4.797, -87.881, 119.453, -3.645, 23.473, 8.184]
  MoveL 434 to (-826.52, 135.51, -310.07) mm, rotated rx 0 ry 55.74 rz 88.34 deg; joints [4.756, -87.627, 118.807, -3.153, 24.575, 7.731]
  MoveL 435 to (-826.52, 130.17, -302.13) mm, rotated rx 0 ry 56.46 rz 88.26 deg; joints [4.713, -87.349, 118.127, -2.674, 25.68, 7.298]
  MoveL 436 to (-826.52, 124.32, -293.18) mm, rotated rx 0 ry 57.2 rz 88.17 deg; joints [4.665, -87.036, 117.383, -2.192, 26.838, 6.869]
  MoveL 437 to (-826.52, 118, -283.24) mm, rotated rx 0 ry 57.97 rz 88.06 deg; joints [4.613, -86.684, 116.575, -1.718, 28.045, 6.453]
  MoveL 438 to (-826.52, 111.28, -272.34) mm, rotated rx 0 ry 58.76 rz 87.95 deg; joints [4.558, -86.295, 115.706, -1.262, 29.298, 6.058]
  MoveL 439 to (-826.52, 104.22, -260.5) mm, rotated rx 0 ry 59.57 rz 87.85 deg; joints [4.502, -85.865, 114.775, -0.837, 30.6, 5.692]
  MoveL 440 to (-826.52, 96.87, -247.77) mm, rotated rx 0 ry 60.45 rz 87.75 deg; joints [4.444, -85.389, 113.773, -0.442, 31.99, 5.352]
  MoveL 441 to (-826.52, 89.3, -234.18) mm, rotated rx 0 ry 61.37 rz 87.66 deg; joints [4.387, -84.869, 112.709, -0.092, 33.442, 5.048]
  MoveL 442 to (-826.52, 81.57, -219.74) mm, rotated rx 0 ry 62.32 rz 87.59 deg; joints [4.331, -84.304, 111.584, 0.206, 34.949, 4.785]
  MoveL 443 to (-826.52, 73.74, -204.51) mm, rotated rx 0 ry 63.32 rz 87.55 deg; joints [4.278, -83.694, 110.398, 0.448, 36.517, 4.563]
  MoveL 444 to (-826.52, 65.87, -188.51) mm, rotated rx 0 ry 64.34 rz 87.53 deg; joints [4.228, -83.042, 109.16, 0.628, 38.12, 4.385]
  MoveL 445 to (-826.52, 50.77, -155.73) mm, rotated rx 0 ry 66.23 rz 87.62 deg; joints [4.151, -81.696, 106.684, 0.76, 41.138, 4.185]
  MoveL 446 to (-826.52, 36.83, -122.59) mm, rotated rx 0 ry 68.2 rz 87.86 deg; joints [4.1, -80.266, 104.145, 0.657, 44.233, 4.13]
  MoveL 447 to (-826.52, 24.1, -89.04) mm, rotated rx 0 ry 70.26 rz 88.26 deg; joints [4.075, -78.752, 101.541, 0.353, 47.396, 4.184]
  MoveL 448 to (-826.52, 24.1, -89.04) mm, rotated rx 0 ry 70.26 rz 88.26 deg; joints [4.075, -78.752, 101.541, 0.353, 47.396, 4.184]
  MoveL 449 to (-827.4, 20.67, -79.27) mm, rotated rx 0 ry 70.85 rz 88.4 deg; joints [4.05, -78.304, 100.784, 0.24, 48.306, 4.191]
  MoveL 450 to (-830, 17.48, -69.73) mm, rotated rx 0 ry 71.4 rz 88.55 deg; joints [3.986, -77.872, 100.061, 0.13, 49.16, 4.154]
  MoveL 451 to (-834.28, 14.59, -60.72) mm, rotated rx 0 ry 71.89 rz 88.71 deg; joints [3.883, -77.471, 99.393, 0.028, 49.926, 4.075]
  MoveL 452 to (-840.15, 12.08, -52.55) mm, rotated rx 0 ry 72.3 rz 88.85 deg; joints [3.744, -77.118, 98.809, -0.062, 50.57, 3.955]
  MoveL 453 to (-843.65, 10.98, -48.88) mm, rotated rx 0 ry 72.46 rz 88.92 deg; joints [3.662, -76.964, 98.556, -0.1, 50.836, 3.879]
  MoveL 454 to (-847.5, 10, -45.55) mm, rotated rx 0 ry 72.59 rz 88.99 deg; joints [3.571, -76.83, 98.333, -0.132, 51.06, 3.794]
  MoveL 455 to (-851.67, 9.16, -42.62) mm, rotated rx 0 ry 72.69 rz 89.04 deg; joints [3.473, -76.716, 98.145, -0.156, 51.237, 3.698]
  MoveL 456 to (-856.13, 8.45, -40.12) mm, rotated rx 0 ry 72.76 rz 89.09 deg; joints [3.368, -76.624, 97.994, -0.172, 51.365, 3.592]
  MoveL 457 to (-860.86, 7.89, -38.09) mm, rotated rx 0 ry 72.79 rz 89.14 deg; joints [3.256, -76.557, 97.883, -0.177, 51.442, 3.477]
  MoveL 458 to (-865.79, 7.5, -36.58) mm, rotated rx 0 ry 72.78 rz 89.17 deg; joints [3.139, -76.515, 97.814, -0.171, 51.465, 3.352]
  MoveL 459 to (-870.88, 7.27, -35.61) mm, rotated rx 0 ry 72.74 rz 89.19 deg; joints [3.018, -76.5, 97.789, -0.152, 51.435, 3.218]
  MoveL 460 to (-876.05, 7.22, -35.21) mm, rotated rx 0 ry 72.67 rz 89.19 deg; joints [2.893, -76.513, 97.809, -0.12, 51.351, 3.077]
  MoveL 461 to (-881.23, 7.35, -35.39) mm, rotated rx 0 ry 72.56 rz 89.19 deg; joints [2.768, -76.551, 97.872, -0.075, 51.217, 2.93]
  MoveL 462 to (-886.35, 7.66, -36.14) mm, rotated rx 0 ry 72.42 rz 89.18 deg; joints [2.643, -76.616, 97.979, -0.016, 51.036, 2.779]
  MoveL 463 to (-891.34, 8.15, -37.45) mm, rotated rx 0 ry 72.25 rz 89.15 deg; joints [2.52, -76.704, 98.125, 0.055, 50.812, 2.625]
  MoveL 464 to (-896.14, 8.81, -39.28) mm, rotated rx 0 ry 72.07 rz 89.11 deg; joints [2.4, -76.814, 98.308, 0.138, 50.551, 2.47]
  MoveL 465 to (-900.7, 9.64, -41.6) mm, rotated rx 0 ry 71.86 rz 89.06 deg; joints [2.286, -76.944, 98.525, 0.231, 50.257, 2.316]
  MoveL 466 to (-904.97, 10.62, -44.36) mm, rotated rx 0 ry 71.64 rz 89.01 deg; joints [2.177, -77.091, 98.771, 0.332, 49.935, 2.165]
  MoveL 467 to (-908.91, 11.75, -47.52) mm, rotated rx 0 ry 71.41 rz 88.95 deg; joints [2.075, -77.253, 99.043, 0.439, 49.591, 2.018]
  MoveL 468 to (-912.51, 13.01, -51.04) mm, rotated rx 0 ry 71.16 rz 88.88 deg; joints [1.981, -77.427, 99.337, 0.551, 49.228, 1.876]
  MoveL 469 to (-918.55, 15.87, -58.96) mm, rotated rx 0 ry 70.66 rz 88.74 deg; joints [1.82, -77.805, 99.977, 0.782, 48.464, 1.616]
  MoveL 470 to (-922.95, 19.12, -67.78) mm, rotated rx 0 ry 70.16 rz 88.59 deg; joints [1.698, -78.209, 100.667, 1.01, 47.669, 1.395]
  MoveL 471 to (-925.62, 22.62, -77.17) mm, rotated rx 0 ry 69.66 rz 88.45 deg; joints [1.618, -78.626, 101.382, 1.222, 46.868, 1.222]
  MoveL 472 to (-926.52, 26.29, -86.85) mm, rotated rx 0 ry 69.17 rz 88.31 deg; joints [1.584, -79.045, 102.103, 1.407, 46.076, 1.105]
  MoveL 473 to (-926.52, 26.29, -86.85) mm, rotated rx 0 ry 69.17 rz 88.31 deg; joints [1.584, -79.045, 102.103, 1.407, 46.076, 1.105]
  MoveL 474 to (-926.52, 38.04, -116.58) mm, rotated rx 0 ry 67.72 rz 87.98 deg; joints [1.561, -80.295, 104.287, 1.854, 43.691, 0.872]
  MoveL 475 to (-926.52, 50.56, -146.07) mm, rotated rx 0 ry 66.32 rz 87.77 deg; joints [1.559, -81.496, 106.431, 2.149, 41.345, 0.712]
  MoveL 476 to (-926.52, 63.84, -175.38) mm, rotated rx 0 ry 64.97 rz 87.68 deg; joints [1.576, -82.647, 108.534, 2.273, 39.044, 0.643]
  MoveL 477 to (-926.52, 77.73, -204.19) mm, rotated rx 0 ry 63.54 rz 87.72 deg; joints [1.615, -83.762, 110.628, 2.21, 36.636, 0.687]
  MoveL 478 to (-926.52, 92.31, -232.48) mm, rotated rx 0 ry 61.94 rz 87.86 deg; joints [1.671, -84.851, 112.745, 1.972, 34.002, 0.848]
  MoveL 479 to (-926.52, 107.72, -260.37) mm, rotated rx 0 ry 60.22 rz 88.07 deg; joints [1.742, -85.896, 114.871, 1.564, 31.208, 1.133]
  MoveL 480 to (-926.52, 124.23, -288.15) mm, rotated rx 0 ry 58.29 rz 88.32 deg; joints [1.821, -86.911, 117.06, 1.009, 28.105, 1.545]
  MoveL 481 to (-926.52, 142.65, -316.5) mm, rotated rx 0 ry 55.51 rz 88.5 deg; joints [1.899, -87.968, 119.552, 0.395, 23.894, 2.054]
  MoveL 482 to (-926.52, 152.37, -330.16) mm, rotated rx 0 ry 53.58 rz 88.5 deg; joints [1.928, -88.494, 120.941, 0.181, 21.103, 2.275]
  MoveL 483 to (-926.52, 157.28, -336.68) mm, rotated rx 0 ry 52.44 rz 88.45 deg; joints [1.937, -88.748, 121.671, 0.137, 19.487, 2.35]
  MoveL 484 to (-926.52, 162.02, -342.7) mm, rotated rx 0 ry 51.22 rz 88.38 deg; joints [1.942, -88.982, 122.396, 0.157, 17.783, 2.38]
  MoveL 485 to (-926.52, 166.47, -348.12) mm, rotated rx 0 ry 49.98 rz 88.28 deg; joints [1.943, -89.189, 123.094, 0.255, 16.041, 2.352]
  MoveL 486 to (-926.52, 170.6, -352.93) mm, rotated rx 0 ry 48.73 rz 88.15 deg; joints [1.941, -89.367, 123.757, 0.444, 14.303, 2.249]
  MoveL 487 to (-926.52, 174.35, -357.12) mm, rotated rx 0 ry 47.52 rz 88.01 deg; joints [1.935, -89.513, 124.367, 0.736, 12.631, 2.054]
  MoveL 488 to (-926.52, 177.69, -360.69) mm, rotated rx 0 ry 46.4 rz 87.86 deg; joints [1.928, -89.628, 124.913, 1.14, 11.079, 1.753]
  MoveL 489 to (-926.52, 180.56, -363.63) mm, rotated rx 0 ry 44.82 rz 87.44 deg; joints [1.888, -89.74, 125.555, 2.967, 8.967, 0.213]
  MoveL 490 to (-926.52, 183.03, -366.02) mm, rotated rx 0 ry 43.31 rz 86.99 deg; joints [1.843, -89.819, 126.14, 5.973, 6.958, -2.474]
  MoveL 491 to (-926.52, 188.02, -370.44) mm, rotated rx 0 ry 39.93 rz 85.8 deg; joints [1.733, -89.898, 127.374, 30.204, 2.707, -25.845]
  MoveL 492 to (-926.52, 198.88, -378.31) mm, rotated rx 12.07 ry 29.88 rz 105.19 deg; joints [1.441, -89.562, 129.985, 160.736, 9.213, -173.377]
  MoveL 493 to (-926.52, 204.93, -381.75) mm, rotated rx 0 ry 27.95 rz 79.14 deg; joints [1.282, -89.08, 131.211, 164.814, 15.164, -155.106]
  MoveL 494 to (-926.52, 211.53, -384.88) mm, rotated rx 0 ry 24.11 rz 75.62 deg; joints [1.13, -88.398, 132.301, 166.556, 21.032, -153.802]
  MoveL 495 to (-926.52, 218.77, -387.74) mm, rotated rx 0 ry 20.7 rz 71.37 deg; joints [0.994, -87.563, 133.229, 167.504, 26.544, -150.943]
  MoveL 496 to (-926.52, 226.78, -390.34) mm, rotated rx 0 ry 17.82 rz 66.4 deg; joints [0.88, -86.63, 133.994, 168.1, 31.535, -146.984]
  MoveL 497 to (-926.52, 235.65, -392.71) mm, rotated rx 0 ry 15.48 rz 60.84 deg; joints [0.789, -85.645, 134.615, 168.521, 35.943, -142.204]
  MoveL 498 to (-926.52, 245.5, -394.87) mm, rotated rx 0 ry 13.67 rz 54.88 deg; joints [0.717, -84.64, 135.118, 168.847, 39.782, -136.892]
  MoveL 499 to (-926.52, 256.56, -396.86) mm, rotated rx 0 ry 12.29 rz 48.74 deg; joints [0.663, -83.616, 135.535, 169.123, 43.15, -131.31]
  MoveL 500 to (-926.52, 269.05, -398.72) mm, rotated rx 0 ry 11.27 rz 42.69 deg; joints [0.624, -82.566, 135.886, 169.373, 46.132, -125.757]
  MoveL 501 to (-926.52, 269.05, -398.72) mm, rotated rx 0 ry 11.27 rz 42.69 deg; joints [0.624, -82.566, 135.886, 169.373, 46.132, -125.757]
  MoveL 502 to (-927.33, 280.42, -400.02) mm, rotated rx 0 ry 10.65 rz 37.97 deg; joints [0.571, -81.678, 136.13, 169.521, 48.34, -121.382]
  MoveL 503 to (-929.69, 291.65, -400.88) mm, rotated rx 0 ry 10.23 rz 33.97 deg; joints [0.473, -80.842, 136.316, 169.562, 50.193, -117.624]
  MoveL 504 to (-933.5, 302.45, -401.34) mm, rotated rx 0 ry 9.95 rz 30.68 deg; joints [0.33, -80.064, 136.453, 169.509, 51.747, -114.491]
  MoveL 505 to (-938.74, 312.67, -401.41) mm, rotated rx 0 ry 9.77 rz 28.01 deg; joints [0.14, -79.345, 136.548, 169.367, 53.058, -111.906]
  MoveL 506 to (-945.38, 321.97, -401.12) mm, rotated rx 0 ry 9.67 rz 25.88 deg; joints [-0.096, -78.696, 136.606, 169.139, 54.148, -109.803]
  MoveL 507 to (-949.23, 326.18, -400.83) mm, rotated rx 0 ry 9.64 rz 25.01 deg; joints [-0.232, -78.402, 136.621, 168.992, 54.615, -108.91]
  MoveL 508 to (-953.44, 330.03, -400.46) mm, rotated rx 0 ry 9.62 rz 24.24 deg; joints [-0.379, -78.132, 136.627, 168.823, 55.028, -108.115]
  MoveL 509 to (-957.98, 333.44, -399.99) mm, rotated rx 0 ry 9.61 rz 23.59 deg; joints [-0.538, -77.889, 136.625, 168.632, 55.386, -107.412]
  MoveL 510 to (-962.83, 336.35, -399.43) mm, rotated rx 0 ry 9.61 rz 23.05 deg; joints [-0.708, -77.678, 136.613, 168.419, 55.684, -106.8]
  MoveL 511 to (-967.97, 338.66, -398.78) mm, rotated rx 0 ry 9.62 rz 22.61 deg; joints [-0.887, -77.504, 136.592, 168.185, 55.92, -106.277]
  MoveL 512 to (-973.36, 340.3, -398.04) mm, rotated rx 0 ry 9.65 rz 22.29 deg; joints [-1.074, -77.37, 136.562, 167.931, 56.087, -105.843]
  MoveL 513 to (-978.91, 341.18, -397.22) mm, rotated rx 0 ry 9.68 rz 22.07 deg; joints [-1.267, -77.283, 136.523, 167.66, 56.181, -105.501]
  MoveL 514 to (-984.52, 341.23, -396.33) mm, rotated rx 0 ry 9.72 rz 21.97 deg; joints [-1.462, -77.247, 136.476, 167.375, 56.198, -105.254]
  MoveL 515 to (-990.05, 340.44, -395.4) mm, rotated rx 0 ry 9.76 rz 21.99 deg; joints [-1.653, -77.263, 136.421, 167.082, 56.136, -105.107]
  MoveL 516 to (-995.39, 338.81, -394.44) mm, rotated rx 0 ry 9.82 rz 22.12 deg; joints [-1.838, -77.331, 136.36, 166.788, 55.996, -105.06]
  MoveL 517 to (-1000.43, 336.4, -393.48) mm, rotated rx 0 ry 9.88 rz 22.37 deg; joints [-2.011, -77.449, 136.294, 166.496, 55.781, -105.114]
  MoveL 518 to (-1005.08, 333.29, -392.52) mm, rotated rx 0 ry 9.94 rz 22.72 deg; joints [-2.171, -77.612, 136.224, 166.212, 55.499, -105.27]
  MoveL 519 to (-1009.29, 329.6, -391.58) mm, rotated rx 0 ry 10.01 rz 23.19 deg; joints [-2.315, -77.813, 136.15, 165.94, 55.155, -105.526]
  MoveL 520 to (-1013.02, 325.42, -390.68) mm, rotated rx 0 ry 10.08 rz 23.75 deg; joints [-2.443, -78.048, 136.075, 165.681, 54.756, -105.882]
  MoveL 521 to (-1016.28, 320.84, -389.82) mm, rotated rx 0 ry 10.16 rz 24.42 deg; joints [-2.553, -78.312, 135.998, 165.436, 54.306, -106.339]
  MoveL 522 to (-1019.06, 315.93, -388.99) mm, rotated rx 0 ry 10.24 rz 25.2 deg; joints [-2.647, -78.601, 135.919, 165.205, 53.808, -106.901]
  MoveL 523 to (-1023.26, 305.42, -387.46) mm, rotated rx 0 ry 10.42 rz 27.09 deg; joints [-2.786, -79.238, 135.756, 164.785, 52.675, -108.356]
  MoveL 524 to (-1025.72, 294.33, -386.08) mm, rotated rx 0 ry 10.65 rz 29.47 deg; joints [-2.862, -79.938, 135.586, 164.42, 51.362, -110.29]
  MoveL 525 to (-1026.52, 282.93, -384.84) mm, rotated rx 0 ry 10.94 rz 32.4 deg; joints [-2.877, -80.693, 135.404, 164.102, 49.844, -112.777]
  MoveL 526 to (-1026.52, 282.93, -384.84) mm, rotated rx 0 ry 10.94 rz 32.4 deg; joints [-2.877, -80.693, 135.404, 164.102, 49.844, -112.777]
  MoveL 527 to (-1026.52, 269.03, -383.28) mm, rotated rx 0 ry 11.44 rz 36.78 deg; joints [-2.856, -81.665, 135.15, 163.707, 47.684, -116.553]
  MoveL 528 to (-1026.52, 256.47, -381.63) mm, rotated rx 0 ry 12.1 rz 41.59 deg; joints [-2.826, -82.6, 134.863, 163.265, 45.33, -120.705]
  MoveL 529 to (-1026.52, 245.15, -379.88) mm, rotated rx 0 ry 12.98 rz 46.72 deg; joints [-2.786, -83.507, 134.537, 162.757, 42.732, -125.09]
  MoveL 530 to (-1026.52, 234.97, -378.03) mm, rotated rx 0 ry 14.13 rz 52 deg; joints [-2.735, -84.393, 134.161, 162.151, 39.84, -129.506]
  MoveL 531 to (-1026.52, 225.8, -376.05) mm, rotated rx 0 ry 15.6 rz 57.24 deg; joints [-2.669, -85.26, 133.722, 161.4, 36.606, -133.71]
  MoveL 532 to (-1026.52, 217.47, -373.92) mm, rotated rx 0 ry 17.45 rz 62.29 deg; joints [-2.586, -86.111, 133.2, 160.416, 32.962, -137.468]
  MoveL 533 to (-1026.52, 209.87, -371.62) mm, rotated rx 0 ry 19.74 rz 67 deg; joints [-2.482, -86.933, 132.572, 159.056, 28.868, -140.485]
  MoveL 534 to (-1026.52, 202.94, -369.12) mm, rotated rx 0 ry 22.47 rz 71.27 deg; joints [-2.357, -87.701, 131.822, 157.053, 24.335, -142.375]
  MoveL 535 to (-1026.52, 196.6, -366.42) mm, rotated rx 0 ry 25.62 rz 75 deg; joints [-2.211, -88.38, 130.936, 153.86, 19.438, -142.525]
  MoveL 536 to (-1026.52, 190.78, -363.5) mm, rotated rx 0 ry 29.13 rz 78.19 deg; joints [-2.046, -88.93, 129.915, 148.162, 14.347, -139.611]
  MoveL 537 to (-1026.52, 180.46, -356.92) mm, rotated rx 0 ry 36.68 rz 83.03 deg; joints [-1.686, -89.532, 127.557, 104.802, 5.699, -100.284]
  MoveL 538 to (-1026.52, 171.79, -349.63) mm, rotated rx 0 ry 43.6 rz 86.03 deg; joints [-1.365, -89.493, 125.172, 25.313, 8.735, -23.124]
  MoveL 539 to (-1026.52, 164.56, -342.07) mm, rotated rx 0 ry 48.77 rz 87.69 deg; joints [-1.144, -89.118, 123.194, 9.735, 14.908, -8.749]
  MoveL 540 to (-1026.52, 158.43, -334.62) mm, rotated rx 0 ry 51.94 rz 88.41 deg; joints [-1.034, -88.712, 121.791, 5.818, 18.966, -5.339]
  MoveL 541 to (-1026.52, 152.76, -327.16) mm, rotated rx 0 ry 53.57 rz 88.53 deg; joints [-1.011, -88.392, 120.856, 4.93, 21.191, -4.541]
  MoveL 542 to (-1026.52, 141.41, -310.95) mm, rotated rx 0 ry 56.28 rz 88.64 deg; joints [-0.986, -87.707, 119.077, 3.984, 24.974, -3.676]
  MoveL 543 to (-1026.52, 130.03, -293.19) mm, rotated rx 0 ry 58.35 rz 88.6 deg; joints [-0.983, -86.991, 117.411, 3.643, 27.991, -3.32]
  MoveL 544 to (-1026.52, 118.62, -274.07) mm, rotated rx 0 ry 59.95 rz 88.47 deg; joints [-0.994, -86.258, 115.821, 3.593, 30.449, -3.194]
  MoveL 545 to (-1026.52, 107.25, -253.88) mm, rotated rx 0 ry 61.25 rz 88.31 deg; joints [-1.01, -85.506, 114.264, 3.658, 32.564, -3.157]
  MoveL 546 to (-1026.52, 95.98, -232.81) mm, rotated rx 0 ry 62.45 rz 88.14 deg; joints [-1.026, -84.719, 112.695, 3.739, 34.544, -3.133]
  MoveL 547 to (-1026.52, 84.71, -210.7) mm, rotated rx 0 ry 63.54 rz 88 deg; joints [-1.038, -83.891, 111.094, 3.789, 36.42, -3.091]
  MoveL 548 to (-1026.52, 73.34, -187.34) mm, rotated rx 0 ry 64.59 rz 87.91 deg; joints [-1.041, -83.014, 109.438, 3.775, 38.246, -3.01]
  MoveL 549 to (-1026.52, 61.77, -162.52) mm, rotated rx 0 ry 65.41 rz 87.88 deg; joints [-1.033, -82.114, 107.77, 3.675, 39.833, -2.884]
  MoveL 550 to (-1026.52, 50.13, -136.57) mm, rotated rx 0 ry 66.3 rz 87.96 deg; joints [-1.01, -81.15, 106.009, 3.437, 41.509, -2.678]
  MoveL 551 to (-1026.52, 28.35, -84.78) mm, rotated rx 0 ry 68.13 rz 88.4 deg; joints [-0.917, -79.157, 102.444, 2.587, 44.886, -2.089]
  MoveL 552 to (-1026.52, 28.35, -84.78) mm, rotated rx 0 ry 68.13 rz 88.4 deg; joints [-0.917, -79.157, 102.444, 2.587, 44.886, -2.089]
  MoveL 553 to (-1027.41, 24.59, -75.28) mm, rotated rx 0 ry 68.46 rz 88.53 deg; joints [-0.915, -78.784, 101.788, 2.392, 45.493, -1.988]
  MoveL 554 to (-1030.05, 21.03, -66.02) mm, rotated rx 0 ry 68.75 rz 88.66 deg; joints [-0.956, -78.422, 101.157, 2.211, 46.052, -1.942]
  MoveL 555 to (-1034.38, 17.76, -57.32) mm, rotated rx 0 ry 68.99 rz 88.81 deg; joints [-1.038, -78.084, 100.574, 2.049, 46.537, -1.951]
  MoveL 556 to (-1040.32, 14.88, -49.49) mm, rotated rx 0 ry 69.16 rz 88.94 deg; joints [-1.16, -77.786, 100.061, 1.918, 46.924, -2.018]
  MoveL 557 to (-1043.85, 13.62, -45.99) mm, rotated rx 0 ry 69.22 rz 89.01 deg; joints [-1.236, -77.655, 99.838, 1.866, 47.075, -2.075]
  MoveL 558 to (-1047.72, 12.49, -42.85) mm, rotated rx 0 ry 69.26 rz 89.07 deg; joints [-1.32, -77.54, 99.642, 1.827, 47.194, -2.146]
  MoveL 559 to (-1051.91, 11.51, -40.08) mm, rotated rx 0 ry 69.28 rz 89.12 deg; joints [-1.413, -77.44, 99.474, 1.8, 47.28, -2.232]
  MoveL 560 to (-1056.38, 10.69, -37.73) mm, rotated rx 0 ry 69.27 rz 89.17 deg; joints [-1.515, -77.358, 99.337, 1.788, 47.332, -2.334]
  MoveL 561 to (-1061.09, 10.04, -35.84) mm, rotated rx 0 ry 69.25 rz 89.21 deg; joints [-1.624, -77.295, 99.233, 1.791, 47.349, -2.451]
  MoveL 562 to (-1066, 9.57, -34.44) mm, rotated rx 0 ry 69.2 rz 89.24 deg; joints [-1.739, -77.252, 99.163, 1.811, 47.332, -2.582]
  MoveL 563 to (-1071.04, 9.3, -33.55) mm, rotated rx 0 ry 69.14 rz 89.25 deg; joints [-1.859, -77.228, 99.128, 1.849, 47.282, -2.727]
  MoveL 564 to (-1076.16, 9.23, -33.2) mm, rotated rx 0 ry 69.06 rz 89.26 deg; joints [-1.984, -77.225, 99.13, 1.904, 47.201, -2.883]
  MoveL 565 to (-1081.28, 9.37, -33.38) mm, rotated rx 0 ry 68.96 rz 89.26 deg; joints [-2.11, -77.242, 99.167, 1.975, 47.091, -3.05]
  MoveL 566 to (-1086.34, 9.71, -34.1) mm, rotated rx 0 ry 68.86 rz 89.25 deg; joints [-2.238, -77.278, 99.238, 2.063, 46.955, -3.225]
  MoveL 567 to (-1091.29, 10.25, -35.33) mm, rotated rx 0 ry 68.74 rz 89.23 deg; joints [-2.365, -77.333, 99.342, 2.165, 46.796, -3.407]
  MoveL 568 to (-1096.06, 10.99, -37.05) mm, rotated rx 0 ry 68.62 rz 89.19 deg; joints [-2.489, -77.404, 99.477, 2.28, 46.618, -3.592]
  MoveL 569 to (-1100.59, 11.92, -39.24) mm, rotated rx 0 ry 68.5 rz 89.15 deg; joints [-2.61, -77.492, 99.639, 2.406, 46.425, -3.778]
  MoveL 570 to (-1104.85, 13.02, -41.86) mm, rotated rx 0 ry 68.37 rz 89.11 deg; joints [-2.726, -77.593, 99.827, 2.54, 46.217, -3.964]
  MoveL 571 to (-1108.81, 14.28, -44.87) mm, rotated rx 0 ry 68.24 rz 89.06 deg; joints [-2.836, -77.708, 100.039, 2.68, 45.999, -4.147]
  MoveL 572 to (-1112.41, 15.68, -48.22) mm, rotated rx 0 ry 68.11 rz 89 deg; joints [-2.939, -77.834, 100.27, 2.824, 45.774, -4.326]
  MoveL 573 to (-1118.49, 18.87, -55.83) mm, rotated rx 0 ry 67.85 rz 88.88 deg; joints [-3.12, -78.114, 100.784, 3.115, 45.305, -4.66]
  MoveL 574 to (-1122.92, 22.45, -64.34) mm, rotated rx 0 ry 67.61 rz 88.75 deg; joints [-3.262, -78.422, 101.347, 3.395, 44.826, -4.954]
  MoveL 575 to (-1125.62, 26.29, -73.47) mm, rotated rx 0 ry 67.38 rz 88.63 deg; joints [-3.363, -78.75, 101.944, 3.653, 44.344, -5.196]
  MoveL 576 to (-1126.52, 30.26, -82.88) mm, rotated rx 0 ry 67.17 rz 88.52 deg; joints [-3.419, -79.086, 102.554, 3.877, 43.87, -5.377]
  MoveL 577 to (-1126.52, 30.26, -82.88) mm, rotated rx 0 ry 67.17 rz 88.52 deg; joints [-3.419, -79.086, 102.554, 3.877, 43.87, -5.377]
  MoveL 578 to (-1126.52, 45.07, -117.4) mm, rotated rx 0 ry 66.4 rz 88.23 deg; joints [-3.522, -80.313, 104.781, 4.513, 42.145, -5.873]
  MoveL 579 to (-1126.52, 60.46, -151.99) mm, rotated rx 0 ry 65.64 rz 88.13 deg; joints [-3.6, -81.52, 106.992, 4.92, 40.404, -6.263]
  MoveL 580 to (-1126.52, 67.74, -167.94) mm, rotated rx 0 ry 65.3 rz 88.14 deg; joints [-3.627, -82.068, 108.004, 5.028, 39.602, -6.4]
  MoveL 581 to (-1126.52, 74.45, -182.4) mm, rotated rx 0 ry 64.99 rz 88.18 deg; joints [-3.647, -82.561, 108.918, 5.082, 38.871, -6.501]
  MoveL 582 to (-1126.52, 86.69, -208.18) mm, rotated rx 0 ry 64.13 rz 88.32 deg; joints [-3.676, -83.483, 110.646, 5.153, 37.202, -6.687]
  MoveL 583 to (-1126.52, 99.64, -234.22) mm, rotated rx 0 ry 62.98 rz 88.51 deg; joints [-3.7, -84.44, 112.48, 5.22, 35.164, -6.895]
  MoveL 584 to (-1126.52, 113.16, -259.93) mm, rotated rx 0 ry 61.48 rz 88.72 deg; joints [-3.725, -85.41, 114.403, 5.373, 32.715, -7.19]
  MoveL 585 to (-1126.52, 120.02, -272.33) mm, rotated rx 0 ry 60.6 rz 88.81 deg; joints [-3.741, -85.888, 115.383, 5.533, 31.332, -7.406]
  MoveL 586 to (-1126.52, 126.85, -284.2) mm, rotated rx 0 ry 59.55 rz 88.87 deg; joints [-3.762, -86.362, 116.388, 5.812, 29.755, -7.722]
  MoveL 587 to (-1126.52, 133.45, -295.16) mm, rotated rx 0 ry 58.32 rz 88.89 deg; joints [-3.789, -86.821, 117.399, 6.257, 27.989, -8.175]
  MoveL 588 to (-1126.52, 139.58, -304.87) mm, rotated rx 0 ry 56.96 rz 88.87 deg; joints [-3.823, -87.245, 118.38, 6.901, 26.094, -8.796]
  MoveL 589 to (-1126.52, 145.01, -312.96) mm, rotated rx 0 ry 55.07 rz 88.61 deg; joints [-3.896, -87.667, 119.435, 8.422, 23.644, -10.126]
  MoveL 590 to (-1126.52, 149.7, -319.34) mm, rotated rx 0 ry 52.25 rz 87.9 deg; joints [-4.04, -88.103, 120.673, 12.023, 20.228, -13.216]
  MoveL 591 to (-1126.52, 154.39, -325.05) mm, rotated rx 0 ry 48.79 rz 86.86 deg; joints [-4.227, -88.498, 122.054, 18.737, 16.215, -19.158]
  MoveL 592 to (-1126.52, 159.29, -330.26) mm, rotated rx 0 ry 44.71 rz 85.4 deg; joints [-4.455, -88.798, 123.566, 32.549, 11.953, -31.859]
  MoveL 593 to (-1126.52, 164.51, -335.02) mm, rotated rx 0 ry 40.21 rz 83.47 deg; joints [-4.712, -88.928, 125.139, 62.292, 8.831, -60.068]
  MoveL 594 to (-1126.52, 170.15, -339.35) mm, rotated rx 0 ry 35.52 rz 80.98 deg; joints [-4.977, -88.831, 126.683, 103.804, 9.563, -99.534]
  MoveL 595 to (-1126.52, 176.31, -343.32) mm, rotated rx 0 ry 30.92 rz 77.86 deg; joints [-5.234, -88.483, 128.115, 129.219, 13.879, -122.291]
  MoveL 596 to (-1126.52, 183.11, -346.94) mm, rotated rx 0 ry 26.67 rz 74.05 deg; joints [-5.466, -87.903, 129.378, 141.139, 19.348, -130.859]
  MoveL 597 to (-1126.52, 190.67, -350.24) mm, rotated rx 0 ry 22.94 rz 69.53 deg; joints [-5.663, -87.144, 130.443, 147.347, 24.822, -132.99]
  MoveL 598 to (-1126.52, 199.08, -353.26) mm, rotated rx 0 ry 19.83 rz 64.36 deg; joints [-5.823, -86.268, 131.318, 150.999, 29.875, -131.881]
  MoveL 599 to (-1126.52, 208.45, -356.02) mm, rotated rx 0 ry 17.35 rz 58.68 deg; joints [-5.948, -85.328, 132.027, 153.356, 34.362, -128.937]
  MoveL 600 to (-1126.52, 218.92, -358.56) mm, rotated rx 0 ry 15.44 rz 52.71 deg; joints [-6.045, -84.356, 132.604, 154.993, 38.28, -124.95]
  MoveL 601 to (-1126.52, 230.72, -360.91) mm, rotated rx 0 ry 13.99 rz 46.67 deg; joints [-6.118, -83.356, 133.085, 156.212, 41.718, -120.448]
  MoveL 602 to (-1126.52, 244.04, -363.11) mm, rotated rx 0 ry 12.93 rz 40.84 deg; joints [-6.173, -82.328, 133.493, 157.169, 44.747, -115.87]
  MoveL 603 to (-1126.52, 259.05, -365.16) mm, rotated rx 0 ry 12.17 rz 35.45 deg; joints [-6.213, -81.263, 133.846, 157.954, 47.445, -111.556]
  MoveL 604 to (-1126.52, 275.9, -367.09) mm, rotated rx 0 ry 11.62 rz 30.68 deg; joints [-6.241, -80.146, 134.156, 158.625, 49.888, -107.724]
  MoveL 605 to (-1126.52, 275.9, -367.09) mm, rotated rx 0 ry 11.62 rz 30.68 deg; joints [-6.241, -80.146, 134.156, 158.625, 49.888, -107.724]
  MoveL 606 to (-1127.31, 287.43, -368.1) mm, rotated rx 0 ry 11.37 rz 28.02 deg; joints [-6.281, -79.407, 134.321, 158.961, 51.32, -105.586]
  MoveL 607 to (-1129.61, 298.76, -368.71) mm, rotated rx 0 ry 11.19 rz 25.77 deg; joints [-6.366, -78.684, 134.441, 159.172, 52.596, -103.759]
  MoveL 608 to (-1133.35, 309.72, -368.95) mm, rotated rx 0 ry 11.06 rz 23.9 deg; joints [-6.497, -77.983, 134.52, 159.27, 53.73, -102.214]
  MoveL 609 to (-1138.5, 320.09, -368.82) mm, rotated rx 0 ry 10.98 rz 22.36 deg; joints [-6.671, -77.315, 134.558, 159.263, 54.728, -100.915]
  MoveL 610 to (-1145.03, 329.59, -368.32) mm, rotated rx 0 ry 10.94 rz 21.12 deg; joints [-6.89, -76.692, 134.556, 159.156, 55.591, -99.829]
  MoveL 611 to (-1148.82, 333.92, -367.94) mm, rotated rx 0 ry 10.93 rz 20.59 deg; joints [-7.016, -76.403, 134.541, 159.064, 55.97, -99.354]
  MoveL 612 to (-1152.95, 337.9, -367.46) mm, rotated rx 0 ry 10.93 rz 20.14 deg; joints [-7.153, -76.132, 134.515, 158.948, 56.311, -98.922]
  MoveL 613 to (-1157.43, 341.47, -366.88) mm, rotated rx 0 ry 10.94 rz 19.74 deg; joints [-7.3, -75.882, 134.48, 158.805, 56.612, -98.529]
  MoveL 614 to (-1162.22, 344.55, -366.21) mm, rotated rx 0 ry 10.95 rz 19.41 deg; joints [-7.458, -75.658, 134.434, 158.638, 56.868, -98.173]
  MoveL 615 to (-1167.32, 347.06, -365.43) mm, rotated rx 0 ry 10.97 rz 19.14 deg; joints [-7.625, -75.465, 134.378, 158.444, 57.077, -97.855]
  MoveL 616 to (-1172.67, 348.92, -364.57) mm, rotated rx 0 ry 10.99 rz 18.93 deg; joints [-7.8, -75.306, 134.312, 158.226, 57.232, -97.574]
  MoveL 617 to (-1178.2, 350.04, -363.62) mm, rotated rx 0 ry 11.02 rz 18.79 deg; joints [-7.98, -75.188, 134.237, 157.985, 57.328, -97.331]
  MoveL 618 to (-1183.82, 350.34, -362.6) mm, rotated rx 0 ry 11.06 rz 18.72 deg; joints [-8.162, -75.116, 134.154, 157.724, 57.362, -97.13]
  MoveL 619 to (-1189.4, 349.79, -361.53) mm, rotated rx 0 ry 11.1 rz 18.72 deg; joints [-8.343, -75.092, 134.064, 157.448, 57.331, -96.972]
  MoveL 620 to (-1194.83, 348.36, -360.43) mm, rotated rx 0 ry 11.15 rz 18.8 deg; joints [-8.518, -75.118, 133.969, 157.162, 57.234, -96.862]
  MoveL 621 to (-1199.95, 346.13, -359.33) mm, rotated rx 0 ry 11.2 rz 18.94 deg; joints [-8.683, -75.192, 133.872, 156.873, 57.076, -96.801]
  MoveL 622 to (-1204.71, 343.15, -358.25) mm, rotated rx 0 ry 11.25 rz 19.16 deg; joints [-8.835, -75.311, 133.774, 156.584, 56.861, -96.791]
  MoveL 623 to (-1209.01, 339.54, -357.2) mm, rotated rx 0 ry 11.31 rz 19.44 deg; joints [-8.972, -75.47, 133.676, 156.301, 56.594, -96.833]
  MoveL 624 to (-1212.83, 335.41, -356.2) mm, rotated rx 0 ry 11.36 rz 19.78 deg; joints [-9.093, -75.662, 133.581, 156.026, 56.283, -96.93]
  MoveL 625 to (-1216.16, 330.83, -355.25) mm, rotated rx 0 ry 11.42 rz 20.19 deg; joints [-9.198, -75.884, 133.488, 155.761, 55.932, -97.081]
  MoveL 626 to (-1219.01, 325.91, -354.37) mm, rotated rx 0 ry 11.47 rz 20.65 deg; joints [-9.287, -76.131, 133.398, 155.506, 55.545, -97.288]
  MoveL 627 to (-1221.37, 320.72, -353.54) mm, rotated rx 0 ry 11.53 rz 21.19 deg; joints [-9.36, -76.398, 133.31, 155.263, 55.127, -97.554]
  MoveL 628 to (-1223.26, 315.33, -352.78) mm, rotated rx 0 ry 11.6 rz 21.78 deg; joints [-9.418, -76.682, 133.226, 155.031, 54.68, -97.88]
  MoveL 629 to (-1225.72, 304.15, -351.43) mm, rotated rx 0 ry 11.73 rz 23.17 deg; joints [-9.49, -77.291, 133.067, 154.599, 53.705, -98.726]
  MoveL 630 to (-1226.52, 292.69, -350.3) mm, rotated rx 0 ry 11.88 rz 24.84 deg; joints [-9.507, -77.942, 132.917, 154.204, 52.625, -99.855]
  MoveL 631 to (-1226.52, 292.69, -350.3) mm, rotated rx 0 ry 11.88 rz 24.84 deg; joints [-9.507, -77.942, 132.917, 154.204, 52.625, -99.855]
  MoveL 632 to (-1226.52, 280.99, -349.22) mm, rotated rx 0 ry 12.06 rz 26.87 deg; joints [-9.495, -78.628, 132.761, 153.797, 51.418, -101.291]
  MoveL 633 to (-1226.52, 269.99, -348.11) mm, rotated rx 0 ry 12.28 rz 29.1 deg; joints [-9.482, -79.288, 132.594, 153.362, 50.168, -102.913]
  MoveL 634 to (-1226.52, 259.66, -346.96) mm, rotated rx 0 ry 12.55 rz 31.55 deg; joints [-9.465, -79.923, 132.417, 152.893, 48.864, -104.718]
  MoveL 635 to (-1226.52, 249.96, -345.78) mm, rotated rx 0 ry 12.87 rz 34.21 deg; joints [-9.446, -80.539, 132.228, 152.383, 47.492, -106.694]
  MoveL 636 to (-1226.52, 240.88, -344.55) mm, rotated rx 0 ry 13.26 rz 37.07 deg; joints [-9.422, -81.138, 132.025, 151.821, 46.041, -108.821]
  MoveL 637 to (-1226.52, 232.38, -343.28) mm, rotated rx 0 ry 13.74 rz 40.11 deg; joints [-9.394, -81.723, 131.806, 151.194, 44.497, -111.065]
  MoveL 638 to (-1226.52, 224.43, -341.96) mm, rotated rx 0 ry 14.31 rz 43.31 deg; joints [-9.361, -82.295, 131.569, 150.487, 42.847, -113.38]
  MoveL 639 to (-1226.52, 217, -340.59) mm, rotated rx 0 ry 14.99 rz 46.63 deg; joints [-9.322, -82.858, 131.311, 149.678, 41.077, -115.706]
  MoveL 640 to (-1226.52, 203.6, -337.68) mm, rotated rx 0 ry 16.76 rz 53.42 deg; joints [-9.223, -83.956, 130.715, 147.636, 37.127, -120.075]
  MoveL 641 to (-1226.52, 191.9, -334.53) mm, rotated rx 0 ry 19.18 rz 60.09 deg; joints [-9.088, -85.013, 129.979, 144.702, 32.56, -123.411]
  MoveL 642 to (-1226.52, 181.59, -331.05) mm, rotated rx 0 ry 22.4 rz 66.33 deg; joints [-8.907, -86.01, 129.05, 140.121, 27.32, -124.631]
  MoveL 643 to (-1226.52, 172.49, -327.21) mm, rotated rx 0 ry 26.45 rz 71.85 deg; joints [-8.669, -86.882, 127.88, 132.286, 21.581, -121.847]
  MoveL 644 to (-1226.52, 164.46, -322.96) mm, rotated rx 0 ry 31.27 rz 76.51 deg; joints [-8.375, -87.543, 126.445, 117.506, 15.989, -111.232]
  MoveL 645 to (-1226.52, 157.33, -318.27) mm, rotated rx 0 ry 36.62 rz 80.28 deg; joints [-8.035, -87.908, 124.77, 89.453, 12.236, -86.459]
  MoveL 646 to (-1226.52, 150.94, -313.08) mm, rotated rx 0 ry 42.14 rz 83.24 deg; joints [-7.673, -87.943, 122.936, 53.667, 12.715, -53.162]
  MoveL 647 to (-1226.52, 145.13, -307.34) mm, rotated rx 0 ry 47.42 rz 85.49 deg; joints [-7.32, -87.683, 121.07, 30.128, 16.636, -31.449]
  MoveL 648 to (-1226.52, 139.77, -301.01) mm, rotated rx 0 ry 52.08 rz 87.13 deg; joints [-7.008, -87.224, 119.305, 18.265, 21.374, -20.875]
  MoveL 649 to (-1226.52, 134.71, -294.03) mm, rotated rx 0 ry 55.88 rz 88.26 deg; joints [-6.757, -86.676, 117.737, 12.134, 25.632, -15.608]
  MoveL 650 to (-1226.52, 132.18, -290.18) mm, rotated rx 0 ry 57.47 rz 88.68 deg; joints [-6.654, -86.39, 117.025, 10.191, 27.483, -13.975]
  MoveL 651 to (-1226.52, 129.41, -285.71) mm, rotated rx 0 ry 58.95 rz 89.02 deg; joints [-6.561, -86.083, 116.31, 8.65, 29.242, -12.689]
  MoveL 652 to (-1226.52, 126.2, -280.22) mm, rotated rx 0 ry 60.18 rz 89.24 deg; joints [-6.488, -85.766, 115.611, 7.596, 30.778, -11.796]
  MoveL 653 to (-1226.52, 122.31, -273.33) mm, rotated rx 0 ry 60.91 rz 89.22 deg; joints [-6.457, -85.473, 114.993, 7.251, 31.811, -11.443]
  MoveL 654 to (-1226.52, 105.78, -242.04) mm, rotated rx 0 ry 63.23 rz 89.01 deg; joints [-6.356, -84.228, 112.496, 6.473, 35.357, -10.524]
  MoveL 655 to (-1226.52, 90.3, -210.31) mm, rotated rx 0 ry 64.64 rz 88.74 deg; joints [-6.282, -83.059, 110.264, 6.24, 37.844, -10.08]
  MoveL 656 to (-1226.52, 82.99, -194.71) mm, rotated rx 0 ry 65.16 rz 88.62 deg; joints [-6.248, -82.502, 109.222, 6.177, 38.854, -9.917]
  MoveL 657 to (-1226.52, 79.58, -187.33) mm, rotated rx 0 ry 65.33 rz 88.57 deg; joints [-6.232, -82.251, 108.754, 6.163, 39.243, -9.856]
  MoveL 658 to (-1226.52, 76.42, -180.44) mm, rotated rx 0 ry 65.41 rz 88.52 deg; joints [-6.217, -82.029, 108.344, 6.168, 39.512, -9.816]
  MoveL 659 to (-1226.52, 73.56, -174.18) mm, rotated rx 0 ry 65.48 rz 88.49 deg; joints [-6.204, -81.829, 107.971, 6.165, 39.751, -9.776]
  MoveL 660 to (-1226.52, 71.07, -168.7) mm, rotated rx 0 ry 65.53 rz 88.47 deg; joints [-6.191, -81.653, 107.646, 6.158, 39.957, -9.739]
  MoveL 661 to (-1226.52, 66.71, -159.11) mm, rotated rx 0 ry 65.63 rz 88.43 deg; joints [-6.168, -81.346, 107.077, 6.131, 40.314, -9.666]
  MoveL 662 to (-1226.52, 49.51, -120.84) mm, rotated rx 0 ry 65.98 rz 88.43 deg; joints [-6.057, -80.114, 104.797, 5.848, 41.699, -9.279]
  MoveL 663 to (-1226.52, 32.23, -81.76) mm, rotated rx 0 ry 66.32 rz 88.67 deg; joints [-5.913, -78.85, 102.458, 5.254, 43.053, -8.734]
  MoveL 664 to (-1226.52, 32.23, -81.76) mm, rotated rx 0 ry 66.32 rz 88.67 deg; joints [-5.913, -78.85, 102.458, 5.254, 43.053, -8.734]
  MoveL 665 to (-1227.42, 28.19, -72.48) mm, rotated rx 0 ry 66.38 rz 88.76 deg; joints [-5.896, -78.547, 101.901, 5.082, 43.353, -8.615]
  MoveL 666 to (-1230.09, 24.3, -63.47) mm, rotated rx 0 ry 66.41 rz 88.87 deg; joints [-5.922, -78.249, 101.36, 4.926, 43.615, -8.554]
  MoveL 667 to (-1234.47, 20.71, -55.04) mm, rotated rx 0 ry 66.41 rz 88.99 deg; joints [-5.992, -77.969, 100.857, 4.796, 43.823, -8.557]
  MoveL 668 to (-1240.47, 17.51, -47.5) mm, rotated rx 0 ry 66.36 rz 89.1 deg; joints [-6.104, -77.717, 100.41, 4.704, 43.966, -8.628]
  MoveL 669 to (-1244.03, 16.1, -44.16) mm, rotated rx 0 ry 66.33 rz 89.15 deg; joints [-6.175, -77.605, 100.213, 4.676, 44.01, -8.689]
  MoveL 670 to (-1247.92, 14.84, -41.16) mm, rotated rx 0 ry 66.28 rz 89.2 deg; joints [-6.256, -77.503, 100.038, 4.66, 44.035, -8.768]
  MoveL 671 to (-1252.12, 13.74, -38.54) mm, rotated rx 0 ry 66.22 rz 89.25 deg; joints [-6.346, -77.414, 99.885, 4.66, 44.042, -8.865]
  MoveL 672 to (-1256.6, 12.82, -36.32) mm, rotated rx 0 ry 66.16 rz 89.29 deg; joints [-6.445, -77.337, 99.756, 4.675, 44.032, -8.979]
  MoveL 673 to (-1261.3, 12.09, -34.55) mm, rotated rx 0 ry 66.09 rz 89.32 deg; joints [-6.551, -77.273, 99.654, 4.705, 44.005, -9.11]
  MoveL 674 to (-1266.19, 11.57, -33.24) mm, rotated rx 0 ry 66.01 rz 89.35 deg; joints [-6.664, -77.224, 99.578, 4.752, 43.963, -9.256]
  MoveL 675 to (-1271.2, 11.26, -32.43) mm, rotated rx 0 ry 65.94 rz 89.36 deg; joints [-6.783, -77.189, 99.53, 4.815, 43.909, -9.416]
  MoveL 676 to (-1276.27, 11.18, -32.11) mm, rotated rx 0 ry 65.86 rz 89.37 deg; joints [-6.906, -77.168, 99.51, 4.893, 43.844, -9.588]
  MoveL 677 to (-1281.35, 11.32, -32.3) mm, rotated rx 0 ry 65.79 rz 89.37 deg; joints [-7.032, -77.162, 99.518, 4.985, 43.77, -9.769]
  MoveL 678 to (-1286.38, 11.68, -32.99) mm, rotated rx 0 ry 65.73 rz 89.36 deg; joints [-7.159, -77.171, 99.553, 5.088, 43.69, -9.959]
  MoveL 679 to (-1291.27, 12.27, -34.17) mm, rotated rx 0 ry 65.67 rz 89.35 deg; joints [-7.286, -77.193, 99.613, 5.202, 43.607, -10.152]
  MoveL 680 to (-1296, 13.07, -35.81) mm, rotated rx 0 ry 65.62 rz 89.32 deg; joints [-7.411, -77.228, 99.699, 5.324, 43.521, -10.348]
  MoveL 681 to (-1300.53, 14.07, -37.9) mm, rotated rx 0 ry 65.57 rz 89.3 deg; joints [-7.534, -77.276, 99.808, 5.452, 43.433, -10.543]
  MoveL 682 to (-1304.78, 15.26, -40.4) mm, rotated rx 0 ry 65.54 rz 89.26 deg; joints [-7.651, -77.335, 99.939, 5.582, 43.347, -10.736]
  MoveL 683 to (-1308.73, 16.63, -43.28) mm, rotated rx 0 ry 65.52 rz 89.22 deg; joints [-7.764, -77.406, 100.09, 5.713, 43.26, -10.923]
  MoveL 684 to (-1312.35, 18.15, -46.52) mm, rotated rx 0 ry 65.51 rz 89.18 deg; joints [-7.869, -77.487, 100.26, 5.843, 43.175, -11.103]
  MoveL 685 to (-1318.44, 21.59, -53.87) mm, rotated rx 0 ry 65.5 rz 89.09 deg; joints [-8.057, -77.676, 100.648, 6.091, 43.01, -11.432]
  MoveL 686 to (-1322.9, 25.44, -62.15) mm, rotated rx 0 ry 65.53 rz 89.01 deg; joints [-8.208, -77.897, 101.089, 6.312, 42.848, -11.712]
  MoveL 687 to (-1325.61, 29.53, -71.04) mm, rotated rx 0 ry 65.58 rz 88.93 deg; joints [-8.318, -78.142, 101.567, 6.497, 42.688, -11.932]
  MoveL 688 to (-1326.52, 33.73, -80.27) mm, rotated rx 0 ry 65.63 rz 88.85 deg; joints [-8.383, -78.406, 102.071, 6.641, 42.527, -12.087]
  MoveL 689 to (-1326.52, 33.73, -80.27) mm, rotated rx 0 ry 65.63 rz 88.85 deg; joints [-8.383, -78.406, 102.071, 6.641, 42.527, -12.087]
  MoveL 690 to (-1326.52, 38.99, -91.89) mm, rotated rx 0 ry 65.71 rz 88.78 deg; joints [-8.435, -78.745, 102.712, 6.781, 42.316, -12.232]
  MoveL 691 to (-1326.52, 43.93, -102.84) mm, rotated rx 0 ry 65.76 rz 88.74 deg; joints [-8.482, -79.066, 103.317, 6.888, 42.104, -12.357]
  MoveL 692 to (-1326.52, 53.31, -123.73) mm, rotated rx 0 ry 65.85 rz 88.71 deg; joints [-8.563, -79.683, 104.472, 7.024, 41.673, -12.563]
  MoveL 693 to (-1326.52, 62.11, -143.38) mm, rotated rx 0 ry 65.92 rz 88.74 deg; joints [-8.632, -80.265, 105.559, 7.072, 41.238, -12.716]
  MoveL 694 to (-1326.52, 66.2, -152.53) mm, rotated rx 0 ry 65.94 rz 88.77 deg; joints [-8.662, -80.538, 106.066, 7.07, 41.024, -12.774]
  MoveL 695 to (-1326.52, 70.04, -161.15) mm, rotated rx 0 ry 65.96 rz 88.81 deg; joints [-8.689, -80.796, 106.544, 7.055, 40.815, -12.822]
  MoveL 696 to (-1326.52, 73.6, -169.13) mm, rotated rx 0 ry 65.97 rz 88.86 deg; joints [-8.713, -81.036, 106.988, 7.031, 40.614, -12.861]
  MoveL 697 to (-1326.52, 76.85, -176.42) mm, rotated rx 0 ry 65.97 rz 88.91 deg; joints [-8.734, -81.256, 107.395, 7.001, 40.421, -12.893]
  MoveL 698 to (-1326.52, 79.75, -182.93) mm, rotated rx 0 ry 65.96 rz 88.96 deg; joints [-8.752, -81.453, 107.759, 6.969, 40.241, -12.919]
  MoveL 699 to (-1326.52, 82.28, -188.57) mm, rotated rx 0 ry 65.95 rz 89.01 deg; joints [-8.767, -81.626, 108.078, 6.938, 40.077, -12.94]
  MoveL 700 to (-1326.52, 84.39, -193.29) mm, rotated rx 0 ry 65.86 rz 89.05 deg; joints [-8.782, -81.783, 108.368, 6.939, 39.855, -12.981]
  MoveL 701 to (-1326.52, 86.14, -197.19) mm, rotated rx 0 ry 65.76 rz 89.08 deg; joints [-8.794, -81.919, 108.619, 6.95, 39.635, -13.024]
  MoveL 702 to (-1326.52, 89.67, -205) mm, rotated rx 0 ry 65.54 rz 89.16 deg; joints [-8.819, -82.192, 109.127, 6.978, 39.174, -13.117]
  MoveL 703 to (-1326.52, 104.68, -237.1) mm, rotated rx 0 ry 64.2 rz 89.46 deg; joints [-8.935, -83.371, 111.347, 7.286, 36.789, -13.674]
  MoveL 704 to (-1326.52, 112.3, -252.5) mm, rotated rx 0 ry 63.06 rz 89.55 deg; joints [-9.014, -84.001, 112.573, 7.791, 35.076, -14.239]
  MoveL 705 to (-1326.52, 120.09, -266.76) mm, rotated rx 0 ry 59.18 rz 88.64 deg; joints [-9.315, -84.945, 114.586, 11.701, 30.556, -17.446]
  MoveL 706 to (-1326.52, 128.8, -279.69) mm, rotated rx 0 ry 52.33 rz 86.48 deg; joints [-9.847, -86.005, 117.424, 22.683, 23.28, -26.717]
